  MoveL 1987 to (-124.69, -0.74, -85.2) mm, rotated rx -55.86 ry 0 rz -88.54 deg; joints [-7.765, -84.155, 125.135, -193.916, 25.687, 224.937, -15.943]
  MoveL 1988 to (-128.3, 0.76, -79.65) mm, rotated rx -58.38 ry 0 rz -89.25 deg; joints [-7.042, -84.625, 125.115, -192.318, 25.683, 221.219, -14.624]
  MoveL 1989 to (-129.64, 1.6, -77.44) mm, rotated rx -59.45 ry 0 rz -89.66 deg; joints [-6.738, -84.814, 125.113, -191.644, 25.683, 219.644, -13.978]
  MoveL 1990 to (-130.13, 1.75, -76.61) mm, rotated rx -59.6 ry 0 rz -89.68 deg; joints [-6.67, -84.846, 125.104, -191.491, 25.683, 219.379, -13.911]
  MoveL 1991 to (-131.58, 1.85, -74.08) mm, rotated rx -60.65 ry 0 rz -89.72 deg; joints [-6.348, -85.031, 125.098, -190.776, 25.683, 217.779, -13.631]
  MoveL 1992 to (-131.68, 2.01, -73.92) mm, rotated rx -61.25 ry 0 rz -90 deg; joints [-6.228, -85.122, 125.098, -190.529, 25.626, 216.991, -13.301]
  MoveL 1993 to (-132.47, 3.26, -72.44) mm, rotated rx -61.9 ry 0 rz -90.54 deg; joints [-6.033, -85.23, 125.095, -190.094, 25.626, 216.013, -12.623]
  MoveL 1994 to (-132.84, 3.74, -71.74) mm, rotated rx -62.11 ry 0 rz -90.68 deg; joints [-5.957, -85.258, 125.083, -189.924, 25.626, 215.669, -12.434]
  MoveL 1995 to (-135.12, 6.38, -67.14) mm, rotated rx -64.03 ry 0 rz -91.76 deg; joints [-5.36, -85.56, 125.068, -188.59, 25.626, 212.719, -10.966]
  MoveL 1996 to (-136.66, 9.17, -63.61) mm, rotated rx -65.62 ry 0 rz -92.98 deg; joints [-4.871, -85.803, 125.068, -187.496, 25.624, 210.269, -9.452]
  MoveL 1997 to (-137.15, 9.63, -62.48) mm, rotated rx -65.62 ry 0 rz -92.98 deg; joints [-4.813, -85.796, 125.038, -187.365, 25.624, 210.166, -9.424]
  MoveL 1998 to (-137.46, 9.66, -61.8) mm, rotated rx -65.75 ry 0 rz -92.99 deg; joints [-4.754, -85.823, 125.037, -187.234, 25.624, 209.938, -9.381]
  MoveL 1999 to (-138.91, 9.39, -58.5) mm, rotated rx -67.12 ry 0 rz -92.84 deg; joints [-4.317, -86.01, 125.026, -186.253, 25.624, 207.801, -9.287]
  MoveL 2000 to (-139.18, 9.27, -57.89) mm, rotated rx -67.23 ry 0 rz -92.81 deg; joints [-4.264, -86.035, 125.026, -186.136, 25.62, 207.599, -9.292]
  MoveL 2001 to (-140.3, 7.99, -55.3) mm, rotated rx -68.09 ry 0 rz -92.35 deg; joints [-3.96, -86.17, 125.028, -185.454, 25.619, 206.193, -9.603]
  MoveL 2002 to (-140.85, 7.99, -53.9) mm, rotated rx -69.03 ry 0 rz -92.23 deg; joints [-3.698, -86.248, 125.002, -184.865, 25.619, 204.788, -9.593]
  MoveL 2003 to (-141.12, 7.84, -53.2) mm, rotated rx -69.03 ry 0 rz -92.23 deg; joints [-3.663, -86.268, 125.002, -184.79, 25.601, 204.728, -9.589]
  MoveL 2004 to (-141.46, 7.5, -52.35) mm, rotated rx -69.38 ry 0 rz -92.09 deg; joints [-3.55, -86.309, 124.998, -184.535, 25.601, 204.182, -9.678]
  MoveL 2005 to (-143.81, 3.71, -45.92) mm, rotated rx -71.82 ry 0 rz -90.62 deg; joints [-2.721, -86.589, 124.971, -182.667, 25.601, 200.243, -10.807]
  MoveL 2006 to (-143.79, 3.76, -45.99) mm, rotated rx -72.66 ry 0 rz -90.59 deg; joints [-2.549, -86.63, 124.954, -182.281, 25.601, 199.099, -10.766]
  MoveL 2007 to (-144.66, 5.18, -43.07) mm, rotated rx -73.82 ry 0 rz -91.15 deg; joints [-2.156, -86.735, 124.931, -181.395, 25.601, 197.222, -10.071]
  MoveL 2008 to (-144.92, 5.41, -42.15) mm, rotated rx -73.82 ry 0 rz -91.15 deg; joints [-2.11, -86.73, 124.913, -181.29, 25.601, 197.138, -10.058]
  MoveL 2009 to (-145.17, 5.36, -41.27) mm, rotated rx -73.92 ry 0 rz -91.15 deg; joints [-2.045, -86.751, 124.913, -181.143, 25.601, 196.921, -10.032]
  MoveL 2010 to (-145.6, 4.99, -39.76) mm, rotated rx -75.16 ry 0 rz -91.08 deg; joints [-1.707, -86.843, 124.903, -180.379, 25.601, 195.072, -9.994]
  MoveL 2011 to (-146.32, 6.55, -36.79) mm, rotated rx -76.33 ry 0 rz -91.69 deg; joints [-1.306, -86.925, 124.872, -179.475, 25.601, 193.173, -9.275]
  MoveL 2012 to (-146.5, 7.02, -35.98) mm, rotated rx -76.68 ry 0 rz -91.89 deg; joints [-1.19, -86.95, 124.865, -179.213, 25.601, 192.612, -9.046]
  MoveL 2013 to (-147.72, 11.76, -29.12) mm, rotated rx -79.41 ry 0 rz -93.75 deg; joints [-0.253, -87.095, 124.783, -177.091, 25.601, 188.16, -6.982]
  MoveL 2014 to (-147.89, 15.71, -26.25) mm, rotated rx -80.75 ry 0 rz -95.48 deg; joints [0.184, -87.181, 124.772, -176.101, 25.601, 186.018, -5.174]
  MoveL 2015 to (-147.93, 16.33, -25.65) mm, rotated rx -80.87 ry 0 rz -95.59 deg; joints [0.239, -87.161, 124.744, -175.974, 25.602, 185.797, -5.057]
  MoveL 2016 to (-148.25, 18.54, -22.05) mm, rotated rx -82.08 ry 0 rz -96.3 deg; joints [0.685, -87.163, 124.666, -174.962, 25.602, 183.763, -4.303]
  MoveL 2017 to (-148.41, 18.88, -20.63) mm, rotated rx -82.08 ry 0 rz -96.3 deg; joints [0.757, -87.157, 124.666, -174.808, 25.658, 183.639, -4.256]
  MoveL 2018 to (-148.62, 18.58, -19.38) mm, rotated rx -82.16 ry 0 rz -96.29 deg; joints [0.84, -87.184, 124.675, -174.62, 25.658, 183.398, -4.252]
  MoveL 2019 to (-148.94, 17.65, -17.69) mm, rotated rx -82.81 ry 0 rz -95.93 deg; joints [1.067, -87.189, 124.644, -174.105, 25.658, 182.333, -4.597]
  MoveL 2020 to (-149.44, 16.99, -13.68) mm, rotated rx -84.63 ry 0 rz -95.55 deg; joints [1.669, -87.189, 124.582, -172.757, 25.74, 179.418, -4.882]
  MoveL 2021 to (-149.51, 16.81, -13.05) mm, rotated rx -84.73 ry 0 rz -95.52 deg; joints [1.722, -87.195, 124.58, -172.636, 25.74, 179.223, -4.914]
  MoveL 2022 to (-149.73, 16.26, -10.96) mm, rotated rx -85.58 ry 0 rz -95.28 deg; joints [2.016, -87.196, 124.561, -171.985, 25.796, 177.841, -5.106]
  MoveL 2023 to (-149.72, 16.22, -11.05) mm, rotated rx -86.54 ry 0 rz -95.58 deg; joints [2.223, -87.245, 124.581, -171.514, 25.796, 176.502, -4.798]
  MoveL 2024 to (-149.59, 18.71, -8.96) mm, rotated rx -87.54 ry 0 rz -97 deg; joints [2.553, -87.314, 124.605, -170.766, 25.796, 174.892, -3.374]
  MoveL 2025 to (-148.52, 25.7, -9.48) mm, rotated rx -87.35 ry 0 rz -99.88 deg; joints [2.485, -87.334, 124.605, -170.895, 25.713, 175.184, -0.55]
  MoveL 2026 to (-148.27, 27.19, -9.1) mm, rotated rx -87.35 ry 0 rz -99.88 deg; joints [2.5, -87.245, 124.553, -170.888, 25.806, 175.184, -0.495]
  MoveL 2027 to (-148.17, 27.92, -8.63) mm, rotated rx -87.52 ry 0 rz -100.16 deg; joints [2.563, -87.245, 124.552, -170.752, 25.823, 174.897, -0.204]
  MoveL 2028 to (-147.29, 33.08, -4.1) mm, rotated rx -89.39 ry 0 rz -102.59 deg; joints [3.204, -87.259, 124.508, -169.293, 25.823, 171.845, 2.19]
  MoveL 2029 to (-147.14, 33.77, -4.05) mm, rotated rx -89.41 ry 0 rz -102.85 deg; joints [3.211, -87.259, 124.508, -169.278, 25.826, 171.813, 2.457]
  MoveL 2030 to (-143.96, 45.19, -6.36) mm, rotated rx -88.52 ry 0 rz -107.6 deg; joints [2.899, -87.293, 124.508, -169.925, 25.639, 173.219, 7.097]
  MoveL 2031 to (-142.1, 50.49, -8.11) mm, rotated rx -87.83 ry 0 rz -109.84 deg; joints [2.657, -87.305, 124.508, -170.441, 25.526, 174.326, 9.262]
  MoveL 2032 to (-141.84, 51.2, -8.22) mm, rotated rx -87.83 ry 0 rz -109.84 deg; joints [2.648, -87.25, 124.46, -170.46, 25.526, 174.342, 9.256]
  MoveL 2033 to (-141.67, 51.67, -8.22) mm, rotated rx -87.83 ry 0 rz -110.03 deg; joints [2.649, -87.25, 124.46, -170.459, 25.526, 174.339, 9.45]
  MoveL 2034 to (-139.95, 56.28, -7.34) mm, rotated rx -88.15 ry 0 rz -111.73 deg; joints [2.763, -87.232, 124.46, -170.228, 25.617, 173.839, 11.21]
  MoveL 2035 to (-137.43, 62.13, -7.66) mm, rotated rx -88.04 ry 0 rz -114.37 deg; joints [2.724, -87.256, 124.46, -170.29, 25.534, 173.991, 13.796]
  MoveL 2036 to (-135.16, 66.76, -9.11) mm, rotated rx -87.45 ry 0 rz -116.54 deg; joints [2.522, -87.278, 124.46, -170.71, 25.401, 174.912, 15.878]
  MoveL 2037 to (-134.83, 67.4, -9.2) mm, rotated rx -87.45 ry 0 rz -116.54 deg; joints [2.515, -87.224, 124.413, -170.727, 25.401, 174.926, 15.872]
  MoveL 2038 to (-134.37, 68.32, -9.18) mm, rotated rx -87.46 ry 0 rz -116.93 deg; joints [2.517, -87.224, 124.413, -170.722, 25.402, 174.914, 16.264]
  MoveL 2039 to (-133.91, 69.25, -8.94) mm, rotated rx -87.46 ry 0 rz -116.93 deg; joints [2.527, -87.162, 124.374, -170.718, 25.458, 174.914, 16.297]
  MoveL 2040 to (-130.27, 76.23, -5.17) mm, rotated rx -88.89 ry 0 rz -119.93 deg; joints [3.033, -87.158, 124.374, -169.615, 25.629, 172.594, 19.389]
  MoveL 2041 to (-129.97, 76.76, -4.82) mm, rotated rx -88.98 ry 0 rz -120.08 deg; joints [3.071, -87.149, 124.374, -169.542, 25.667, 172.446, 19.565]
  MoveL 2042 to (-128.21, 79.76, -2.85) mm, rotated rx -89.74 ry 0 rz -121.42 deg; joints [3.338, -87.142, 124.374, -168.964, 25.756, 171.222, 20.946]
  MoveL 2043 to (-127.99, 80.12, -2.6) mm, rotated rx -89.83 ry 0 rz -121.57 deg; joints [3.37, -87.14, 124.374, -168.895, 25.77, 171.077, 21.109]
  MoveL 2044 to (-126.08, 83.14, -0.8) mm, rotated rx -90.54 ry 0 rz -122.97 deg; joints [3.618, -87.132, 124.374, -168.36, 25.847, 169.935, 22.541]
  MoveL 2045 to (-125.78, 83.59, -0.43) mm, rotated rx -90.54 ry 0 rz -122.97 deg; joints [3.636, -87.11, 124.374, -168.347, 25.919, 169.93, 22.588]
  MoveL 2046 to (-125.56, 83.91, -0.09) mm, rotated rx -90.67 ry 0 rz -123.12 deg; joints [3.682, -87.107, 124.374, -168.249, 25.936, 169.721, 22.74]
  MoveL 2047 to (-125.22, 84.42, 0.77) mm, rotated rx -90.67 ry 0 rz -123.12 deg; joints [3.725, -87.079, 124.374, -168.189, 26.026, 169.679, 22.797]
  MoveL 2048 to (-124.21, 85.78, 4.61) mm, rotated rx -92.13 ry 0 rz -123.76 deg; joints [4.24, -87.039, 124.374, -167.109, 26.227, 167.36, 23.512]
  MoveL 2049 to (-121.27, 89.62, 8.28) mm, rotated rx -93.9 ry 0 rz -125.89 deg; joints [4.815, -87.007, 124.374, -165.88, 26.374, 164.611, 25.651]
  MoveL 2050 to (-120.98, 89.99, 8.63) mm, rotated rx -94.04 ry 0 rz -126.08 deg; joints [4.863, -87.002, 124.374, -165.779, 26.391, 164.389, 25.845]
  MoveL 2051 to (-117.7, 93.74, 12.84) mm, rotated rx -95.6 ry 0 rz -127.92 deg; joints [5.418, -86.916, 124.374, -164.664, 26.653, 161.95, 27.751]
  MoveL 2052 to (-117.06, 94.32, 14.38) mm, rotated rx -95.6 ry 0 rz -127.92 deg; joints [5.493, -86.869, 124.374, -164.564, 26.789, 161.881, 27.828]
  MoveL 2053 to (-116.97, 94.28, 15.39) mm, rotated rx -95.69 ry 0 rz -127.93 deg; joints [5.564, -86.857, 124.374, -164.423, 26.819, 161.68, 27.845]
  MoveL 2054 to (-117, 93.95, 17.04) mm, rotated rx -96.32 ry 0 rz -127.82 deg; joints [5.785, -86.818, 124.374, -163.985, 26.921, 160.707, 27.755]
  MoveL 2055 to (-116.24, 94.53, 18.96) mm, rotated rx -97.62 ry 0 rz -128.26 deg; joints [6.165, -86.752, 124.374, -163.228, 27.078, 158.815, 28.197]
  MoveL 2056 to (-115.96, 94.57, 20.45) mm, rotated rx -97.62 ry 0 rz -128.26 deg; joints [6.239, -86.728, 124.374, -163.097, 27.139, 158.716, 28.219]
  MoveL 2057 to (-116.14, 94.01, 21.92) mm, rotated rx -97.76 ry 0 rz -128.23 deg; joints [6.344, -86.728, 124.378, -162.865, 27.139, 158.394, 28.166]
  MoveL 2058 to (-117.02, 92.32, 24.27) mm, rotated rx -99.1 ry 0 rz -127.32 deg; joints [6.75, -86.614, 124.378, -162.121, 27.401, 156.492, 27.315]
  MoveL 2059 to (-116.98, 92.03, 25.56) mm, rotated rx -99.59 ry 0 rz -127.24 deg; joints [6.921, -86.572, 124.378, -161.796, 27.489, 155.748, 27.239]
  MoveL 2060 to (-117.05, 91.68, 26.5) mm, rotated rx -99.75 ry 0 rz -127.18 deg; joints [7.002, -86.558, 124.378, -161.633, 27.513, 155.466, 27.165]
  MoveL 2061 to (-117.17, 90.63, 29.37) mm, rotated rx -100.93 ry 0 rz -126.8 deg; joints [7.4, -86.447, 124.378, -160.896, 27.731, 153.722, 26.798]
  MoveL 2062 to (-116.45, 90.99, 31.12) mm, rotated rx -102.26 ry 0 rz -127.11 deg; joints [7.769, -86.342, 124.378, -160.212, 27.922, 151.885, 27.102]
  MoveL 2063 to (-116.16, 91, 32.15) mm, rotated rx -102.26 ry 0 rz -127.11 deg; joints [7.82, -86.319, 124.38, -160.136, 27.975, 151.832, 27.119]
  MoveL 2064 to (-116.09, 90.62, 33.43) mm, rotated rx -103.42 ry 0 rz -127.24 deg; joints [8.131, -86.245, 124.38, -159.527, 28.074, 150.208, 27.201]
  MoveL 2065 to (-114.95, 91.49, 34.97) mm, rotated rx -104.01 ry 0 rz -127.78 deg; joints [8.333, -86.178, 124.38, -159.165, 28.189, 149.343, 27.736]
  MoveL 2066 to (-114.26, 91.74, 36.56) mm, rotated rx -104.01 ry 0 rz -127.78 deg; joints [8.41, -86.125, 124.38, -159.076, 28.307, 149.289, 27.785]
  MoveL 2067 to (-114.19, 91.07, 38.4) mm, rotated rx -104.17 ry 0 rz -127.78 deg; joints [8.537, -86.101, 124.38, -158.814, 28.322, 148.929, 27.74]
  MoveL 2068 to (-115.08, 88.3, 42.05) mm, rotated rx -105.61 ry 0 rz -126.7 deg; joints [9.018, -85.922, 124.38, -157.975, 28.604, 146.879, 26.63]
  MoveL 2069 to (-115.21, 87.18, 43.98) mm, rotated rx -106.52 ry 0 rz -126.22 deg; joints [9.3, -85.801, 124.38, -157.51, 28.8, 145.643, 26.156]
  MoveL 2070 to (-115.3, 86.78, 44.52) mm, rotated rx -106.52 ry 0 rz -126.22 deg; joints [9.33, -85.813, 124.395, -157.446, 28.8, 145.594, 26.143]
  MoveL 2071 to (-115.4, 86.48, 44.85) mm, rotated rx -106.64 ry 0 rz -126.1 deg; joints [9.373, -85.795, 124.395, -157.374, 28.825, 145.413, 26.019]
  MoveL 2072 to (-116.47, 83.68, 47.31) mm, rotated rx -107.55 ry 0 rz -125.03 deg; joints [9.681, -85.674, 124.395, -156.836, 28.989, 144.121, 24.905]
  MoveL 2073 to (-116.37, 82.67, 49.3) mm, rotated rx -108.7 ry 0 rz -124.46 deg; joints [10.011, -85.5, 124.395, -156.344, 29.271, 142.643, 24.356]
  MoveL 2074 to (-116.42, 82.21, 49.94) mm, rotated rx -108.7 ry 0 rz -124.46 deg; joints [10.046, -85.509, 124.41, -156.272, 29.271, 142.588, 24.339]
  MoveL 2075 to (-116.6, 81.61, 50.52) mm, rotated rx -108.79 ry 0 rz -124.38 deg; joints [10.095, -85.509, 124.42, -156.168, 29.272, 142.418, 24.231]
  MoveL 2076 to (-117.58, 78.88, 52.54) mm, rotated rx -109.6 ry 0 rz -123.24 deg; joints [10.358, -85.385, 124.42, -155.739, 29.438, 141.308, 23.062]
  MoveL 2077 to (-117.87, 77.18, 54.39) mm, rotated rx -110.51 ry 0 rz -122.43 deg; joints [10.629, -85.234, 124.42, -155.341, 29.661, 140.142, 22.249]
  MoveL 2078 to (-118.08, 76.44, 54.96) mm, rotated rx -110.51 ry 0 rz -122.43 deg; joints [10.664, -85.268, 124.457, -155.268, 29.661, 140.087, 22.234]
  MoveL 2079 to (-118.37, 75.77, 55.27) mm, rotated rx -110.56 ry 0 rz -122.33 deg; joints [10.694, -85.283, 124.477, -155.205, 29.661, 139.985, 22.112]
  MoveL 2080 to (-119.55, 73.3, 56.05) mm, rotated rx -110.88 ry 0 rz -121.21 deg; joints [10.795, -85.231, 124.477, -155.044, 29.728, 139.557, 20.984]
  MoveL 2081 to (-119.75, 72.81, 56.26) mm, rotated rx -110.99 ry 0 rz -120.91 deg; joints [10.828, -85.206, 124.477, -155.012, 29.774, 139.428, 20.698]
  MoveL 2082 to (-120.75, 68.2, 59.75) mm, rotated rx -112.58 ry 0 rz -118.8 deg; joints [11.308, -84.921, 124.477, -154.318, 30.165, 137.402, 18.558]
  MoveL 2083 to (-120.68, 68.16, 59.97) mm, rotated rx -113.09 ry 0 rz -118.48 deg; joints [11.417, -84.827, 124.477, -154.221, 30.331, 136.843, 18.287]
  MoveL 2084 to (-119.88, 66.14, 63.73) mm, rotated rx -114.66 ry 0 rz -117.9 deg; joints [11.903, -84.546, 124.478, -153.484, 30.655, 134.802, 17.604]
  MoveL 2085 to (-119.8, 65.76, 64.28) mm, rotated rx -114.66 ry 0 rz -117.9 deg; joints [11.931, -84.547, 124.487, -153.426, 30.655, 134.76, 17.585]
  MoveL 2086 to (-119.77, 65.42, 64.66) mm, rotated rx -114.82 ry 0 rz -117.78 deg; joints [11.982, -84.516, 124.487, -153.352, 30.689, 134.549, 17.453]
  MoveL 2087 to (-119.95, 61.76, 67.86) mm, rotated rx -116.05 ry 0 rz -116.47 deg; joints [12.369, -84.288, 124.487, -152.752, 30.919, 132.945, 16.034]
  MoveL 2088 to (-120.08, 60.96, 68.35) mm, rotated rx -116.05 ry 0 rz -116.47 deg; joints [12.401, -84.322, 124.526, -152.688, 30.919, 132.897, 16.018]
  MoveL 2089 to (-120.24, 60.38, 68.59) mm, rotated rx -116.15 ry 0 rz -116.22 deg; joints [12.432, -84.303, 124.528, -152.644, 30.944, 132.768, 15.76]
  MoveL 2090 to (-120.98, 56.47, 70.56) mm, rotated rx -117.04 ry 0 rz -114.49 deg; joints [12.694, -84.125, 124.533, -152.289, 31.154, 131.674, 13.981]
  MoveL 2091 to (-118.84, 57.87, 73.02) mm, rotated rx -119.86 ry 0 rz -115.85 deg; joints [13.333, -83.729, 124.533, -151.276, 31.47, 128.216, 15.064]
  MoveL 2092 to (-117.93, 59.53, 73.19) mm, rotated rx -119.93 ry 0 rz -116.68 deg; joints [13.355, -83.714, 124.533, -151.246, 31.484, 128.126, 15.881]
  MoveL 2093 to (-116.76, 60.86, 73.96) mm, rotated rx -119.96 ry 0 rz -116.69 deg; joints [13.377, -83.573, 124.441, -151.246, 31.536, 128.115, 15.894]
  MoveL 2094 to (-115.68, 60.98, 75.54) mm, rotated rx -119.99 ry 0 rz -116.7 deg; joints [13.455, -83.49, 124.441, -151.193, 31.66, 128.079, 15.93]
  MoveL 2095 to (-115.1, 60.65, 76.68) mm, rotated rx -120.49 ry 0 rz -116.68 deg; joints [13.606, -83.402, 124.486, -151.051, 31.848, 127.523, 15.93]
  MoveL 2096 to (-114.03, 60.99, 78.01) mm, rotated rx -121.53 ry 0 rz -117.15 deg; joints [13.854, -83.226, 124.487, -150.681, 31.986, 126.268, 16.281]
  MoveL 2097 to (-113.32, 60.92, 79.08) mm, rotated rx -121.53 ry 0 rz -117.15 deg; joints [13.904, -83.176, 124.487, -150.639, 32.053, 126.256, 16.285]
  MoveL 2098 to (-112.82, 60.37, 80.21) mm, rotated rx -121.68 ry 0 rz -117.14 deg; joints [13.991, -83.14, 124.527, -150.557, 32.161, 126.074, 16.285]
  MoveL 2099 to (-111.85, 57.98, 83.26) mm, rotated rx -123.17 ry 0 rz -116.42 deg; joints [14.421, -82.89, 124.706, -150.237, 32.786, 124.52, 15.672]
  MoveL 2100 to (-109.17, 56.99, 87.4) mm, rotated rx -125.32 ry 0 rz -116.53 deg; joints [14.983, -82.416, 124.727, -149.536, 33.225, 122.038, 15.56]
  MoveL 2101 to (-108.53, 56, 88.83) mm, rotated rx -125.32 ry 0 rz -116.53 deg; joints [15.062, -82.405, 124.784, -149.46, 33.314, 122.01, 15.56]
  MoveL 2102 to (-108.42, 55.2, 89.47) mm, rotated rx -125.62 ry 0 rz -116.21 deg; joints [15.148, -82.344, 124.818, -149.403, 33.443, 121.699, 15.253]
  MoveL 2103 to (-108.75, 53.37, 90.18) mm, rotated rx -125.62 ry 0 rz -116.21 deg; joints [15.205, -82.43, 124.916, -149.296, 33.443, 121.625, 15.22]
  MoveL 2104 to (-112.59, 43.93, 90.56) mm, rotated rx -125.9 ry 0 rz -111.26 deg; joints [15.267, -82.365, 124.924, -149.254, 33.534, 121.353, 10.279]
  MoveL 2105 to (-113.25, 41.96, 90.66) mm, rotated rx -125.95 ry 0 rz -110.24 deg; joints [15.281, -82.349, 124.925, -149.245, 33.554, 121.3, 9.264]
  MoveL 2106 to (-113.56, 41.16, 90.65) mm, rotated rx -125.94 ry 0 rz -109.98 deg; joints [15.283, -82.372, 124.944, -149.241, 33.554, 121.306, 9.002]
  MoveL 2107 to (-113.92, 38.56, 91.31) mm, rotated rx -126.3 ry 0 rz -108.36 deg; joints [15.369, -82.25, 124.944, -149.215, 33.721, 120.978, 7.418]
  MoveL 2108 to (-113.89, 38.54, 91.36) mm, rotated rx -127.16 ry 0 rz -107.51 deg; joints [15.503, -82.032, 124.935, -149.215, 34.026, 120.2, 6.642]
  MoveL 2109 to (-112.68, 37.99, 93.08) mm, rotated rx -128.64 ry 0 rz -107.68 deg; joints [15.823, -81.751, 124.935, -148.756, 34.175, 118.492, 6.59]
  MoveL 2110 to (-110.37, 39.47, 95.21) mm, rotated rx -129.67 ry 0 rz -108.71 deg; joints [16.083, -81.492, 124.935, -148.43, 34.35, 117.33, 7.458]
  MoveL 2111 to (-108.12, 42.41, 96.54) mm, rotated rx -130.58 ry 0 rz -110.86 deg; joints [16.289, -81.324, 124.935, -148.082, 34.373, 116.225, 9.388]
  MoveL 2112 to (-122.31, 47.82, 109.55) mm, rotated rx -130.58 ry 0 rz -110.86 deg; joints [17.015, -81.832, 124.935, -147.724, 35.769, 115.928, 11.072]
  Set speed (1000.0 mm/s)
  MoveL 2113 to (-119.4, 45.41, 113.71) mm, rotated rx -130.84 ry 0 rz -110.73 deg; joints [17.251, -81.623, 124.936, -147.355, 35.823, 115.48, 10.707]
  Set speed (5.0 mm/s)
  MoveL 2114 to (-105.24, 40.05, 100.63) mm, rotated rx -130.84 ry 0 rz -110.73 deg; joints [16.522, -81.126, 124.933, -147.685, 34.394, 115.748, 9.003]
  Set speed (16.7 mm/s)
  MoveL 2115 to (-106.36, 36.25, 100.88) mm, rotated rx -130.97 ry 0 rz -108.71 deg; joints [16.557, -81.101, 124.96, -147.684, 34.47, 115.642, 7.009]
  MoveL 2116 to (-120.67, 41.09, 113.99) mm, rotated rx -130.97 ry 0 rz -108.71 deg; joints [17.287, -81.594, 124.96, -147.351, 35.898, 115.372, 8.711]
  Set speed (1000.0 mm/s)
  MoveL 2117 to (-118.91, 26.12, 120.09) mm, rotated rx -134.04 ry 0 rz -101.52 deg; joints [18.009, -80.673, 124.96, -146.703, 36.636, 112.216, 1.177]
  Set speed (5.0 mm/s)
  MoveL 2118 to (-104.82, 23.25, 106.19) mm, rotated rx -134.04 ry 0 rz -101.52 deg; joints [17.246, -80.243, 124.96, -147.004, 35.105, 112.431, -0.563]
  Set speed (16.7 mm/s)
  MoveL 2119 to (-104.41, 21.99, 106.87) mm, rotated rx -134.42 ry 0 rz -100.89 deg; joints [17.341, -80.162, 125.024, -146.997, 35.3, 112.12, -1.156]
  MoveL 2120 to (-102.69, 19.1, 109.07) mm, rotated rx -135.76 ry 0 rz -99.29 deg; joints [17.628, -79.797, 125.032, -146.697, 35.53, 110.72, -2.963]
  MoveL 2121 to (-102.33, 17.43, 109.68) mm, rotated rx -135.76 ry 0 rz -99.29 deg; joints [17.679, -79.866, 125.12, -146.607, 35.53, 110.665, -3.002]
  MoveL 2122 to (-102.37, 16.88, 109.73) mm, rotated rx -135.79 ry 0 rz -98.98 deg; joints [17.685, -79.858, 125.123, -146.605, 35.542, 110.64, -3.312]
  MoveL 2123 to (-102.11, 14.05, 110.35) mm, rotated rx -136.17 ry 0 rz -97.19 deg; joints [17.764, -79.733, 125.125, -146.565, 35.655, 110.28, -5.136]
  MoveL 2124 to (-102.17, 14.13, 110.3) mm, rotated rx -137.24 ry 0 rz -96.25 deg; joints [17.893, -79.461, 125.103, -146.565, 35.92, 109.327, -6.068]
  MoveL 2125 to (-99.55, 14.42, 112.66) mm, rotated rx -138.55 ry 0 rz -96.54 deg; joints [18.172, -79.095, 125.104, -146.222, 36.066, 107.922, -6.066]
  MoveL 2126 to (-97.81, 15.28, 114.06) mm, rotated rx -139.93 ry 0 rz -97.63 deg; joints [18.416, -78.817, 125.109, -145.827, 36.066, 106.38, -5.341]
  MoveL 2127 to (-95.33, 17.87, 115.77) mm, rotated rx -140.85 ry 0 rz -99.27 deg; joints [18.607, -78.545, 125.109, -145.593, 36.155, 105.406, -3.922]
  MoveL 2128 to (-94.23, 18.44, 116.58) mm, rotated rx -140.85 ry 0 rz -99.27 deg; joints [18.631, -78.445, 125.063, -145.563, 36.162, 105.406, -3.973]
  MoveL 2129 to (-93.66, 18.46, 117.03) mm, rotated rx -140.94 ry 0 rz -99.3 deg; joints [18.662, -78.399, 125.065, -145.533, 36.184, 105.318, -3.973]
  MoveL 2130 to (-92.1, 18.26, 118.3) mm, rotated rx -141.72 ry 0 rz -99.34 deg; joints [18.83, -78.203, 125.157, -145.482, 36.458, 104.634, -3.973]
  MoveL 2131 to (-89.1, 18.17, 120.59) mm, rotated rx -143.24 ry 0 rz -99.6 deg; joints [19.12, -77.798, 125.206, -145.184, 36.651, 103.104, -4.028]
  MoveL 2132 to (-88, 17.68, 121.46) mm, rotated rx -143.24 ry 0 rz -99.6 deg; joints [19.165, -77.76, 125.234, -145.139, 36.684, 103.102, -4.07]
  MoveL 2133 to (-87.65, 17.34, 121.76) mm, rotated rx -143.43 ry 0 rz -99.42 deg; joints [19.203, -77.707, 125.242, -145.105, 36.713, 102.909, -4.29]
  MoveL 2134 to (-87.09, 16.45, 122.28) mm, rotated rx -143.43 ry 0 rz -99.42 deg; joints [19.238, -77.723, 125.287, -145.047, 36.713, 102.882, -4.331]
  MoveL 2135 to (-85.63, 12.54, 123.76) mm, rotated rx -144.42 ry 0 rz -96.96 deg; joints [19.423, -77.447, 125.326, -144.879, 36.855, 101.914, -6.998]
  MoveL 2136 to (-84.87, 11.35, 124.41) mm, rotated rx -144.96 ry 0 rz -95.98 deg; joints [19.509, -77.287, 125.327, -144.803, 36.922, 101.392, -8.081]
  MoveL 2137 to (-84.51, 10.45, 124.72) mm, rotated rx -144.96 ry 0 rz -95.98 deg; joints [19.537, -77.32, 125.377, -144.757, 36.922, 101.369, -8.107]
  MoveL 2138 to (-84.4, 9.74, 124.85) mm, rotated rx -145.01 ry 0 rz -95.79 deg; joints [19.554, -77.33, 125.401, -144.73, 36.922, 101.313, -8.323]
  MoveL 2139 to (-84.29, 8.18, 125.03) mm, rotated rx -145.13 ry 0 rz -94.72 deg; joints [19.577, -77.295, 125.411, -144.721, 36.953, 101.208, -9.404]
  MoveL 2140 to (-84.32, 8.21, 125.03) mm, rotated rx -145.76 ry 0 rz -93.43 deg; joints [19.619, -77.062, 125.321, -144.721, 37.02, 100.633, -10.763]
  MoveL 2141 to (-83.75, 7.93, 125.43) mm, rotated rx -146.04 ry 0 rz -93.26 deg; joints [19.667, -76.985, 125.325, -144.661, 37.034, 100.351, -11.009]
  MoveL 2142 to (-83.33, 7.67, 125.72) mm, rotated rx -146.1 ry 0 rz -93.21 deg; joints [19.689, -76.963, 125.335, -144.629, 37.036, 100.28, -11.104]
  MoveL 2143 to (-82.15, 6.44, 126.56) mm, rotated rx -146.53 ry 0 rz -92.57 deg; joints [19.781, -76.846, 125.374, -144.54, 37.095, 99.856, -11.855]
  MoveL 2144 to (-81.38, 6.16, 127.08) mm, rotated rx -147.23 ry 0 rz -92.07 deg; joints [19.873, -76.66, 125.374, -144.461, 37.162, 99.191, -12.482]
  MoveL 2145 to (-80.87, 5.85, 127.42) mm, rotated rx -147.23 ry 0 rz -92.07 deg; joints [19.894, -76.655, 125.396, -144.439, 37.174, 99.188, -12.502]
  MoveL 2146 to (-80.53, 5.57, 127.65) mm, rotated rx -147.39 ry 0 rz -91.87 deg; joints [19.921, -76.609, 125.399, -144.404, 37.179, 99.02, -12.747]
  MoveL 2147 to (-78.37, 3.33, 129.04) mm, rotated rx -148.32 ry 0 rz -90.39 deg; joints [20.09, -76.357, 125.469, -144.269, 37.316, 98.147, -14.435]
  MoveL 2148 to (-88.88, 3.4, 146.06) mm, rotated rx -148.32 ry 0 rz -90.39 deg; joints [20.959, -76.423, 125.373, -144.051, 39.145, 98.147, -12.66]
  Set speed (1000.0 mm/s)
  MoveL 2149 to (-85.2, 1.1, 148.27) mm, rotated rx -149.48 ry 0 rz -90 deg; joints [21.198, -76.142, 125.476, -143.716, 39.146, 96.927, -13.492]
  Set speed (5.0 mm/s)
  MoveL 2150 to (-75.05, 1.1, 131.04) mm, rotated rx -149.48 ry 0 rz -90 deg; joints [20.326, -76.113, 125.598, -143.946, 37.337, 96.927, -15.233]
  Set speed (16.7 mm/s)
  MoveL 2151 to (-74.99, 0.23, 131.08) mm, rotated rx -149.51 ry 0 rz -89.33 deg; joints [20.33, -76.104, 125.601, -143.946, 37.345, 96.905, -15.908]
  MoveL 2152 to (-75.02, -0.11, 131.07) mm, rotated rx -149.73 ry 0 rz -87.95 deg; joints [20.327, -75.972, 125.518, -143.961, 37.345, 96.712, -17.327]
  MoveL 2153 to (-73.47, -2, 131.92) mm, rotated rx -149.99 ry 0 rz -87.96 deg; joints [20.425, -75.985, 125.642, -143.814, 37.345, 96.396, -17.458]
  MoveL 2154 to (-72.96, -2.95, 132.2) mm, rotated rx -149.99 ry 0 rz -87.96 deg; joints [20.453, -76.026, 125.701, -143.768, 37.345, 96.375, -17.485]
  MoveL 2155 to (-72.33, -5.36, 132.45) mm, rotated rx -150.41 ry 0 rz -85.29 deg; joints [20.493, -75.876, 125.677, -143.768, 37.407, 96.02, -20.214]
  MoveL 2156 to (-71.43, -6.39, 132.9) mm, rotated rx -150.78 ry 0 rz -84.4 deg; joints [20.556, -75.779, 125.726, -143.768, 37.518, 95.721, -21.14]
  MoveL 2157 to (-70.8, -7.68, 133.18) mm, rotated rx -150.78 ry 0 rz -84.4 deg; joints [20.592, -75.844, 125.807, -143.71, 37.518, 95.692, -21.169]
  MoveL 2158 to (-70.31, -9.65, 133.31) mm, rotated rx -150.89 ry 0 rz -82.76 deg; joints [20.611, -75.813, 125.822, -143.71, 37.551, 95.596, -22.816]
  MoveL 2159 to (-70.2, -10.42, 133.32) mm, rotated rx -150.9 ry 0 rz -82.61 deg; joints [20.622, -75.849, 125.856, -143.691, 37.551, 95.576, -22.975]
  MoveL 2160 to (-70.14, -12.43, 133.18) mm, rotated rx -150.79 ry 0 rz -80.96 deg; joints [20.605, -75.876, 125.851, -143.714, 37.551, 95.684, -24.584]
  MoveL 2161 to (-69.55, -15.84, 133.12) mm, rotated rx -150.75 ry 0 rz -77.95 deg; joints [20.593, -75.869, 125.832, -143.731, 37.551, 95.729, -27.582]
  MoveL 2162 to (-69.76, -17.49, 132.81) mm, rotated rx -150.75 ry 0 rz -77.95 deg; joints [20.606, -75.996, 125.923, -143.702, 37.551, 95.697, -27.555]
  MoveL 2163 to (-70.51, -19.37, 132.15) mm, rotated rx -150.01 ry 0 rz -75.72 deg; joints [20.484, -76.103, 125.837, -143.874, 37.551, 96.477, -29.563]
  MoveL 2164 to (-70.5, -20.09, 132.05) mm, rotated rx -149.98 ry 0 rz -75.52 deg; joints [20.485, -76.144, 125.862, -143.87, 37.551, 96.491, -29.754]
  MoveL 2165 to (-70.76, -22.23, 131.56) mm, rotated rx -149.53 ry 0 rz -73.12 deg; joints [20.399, -76.191, 125.788, -143.994, 37.55, 96.98, -32.01]
  MoveL 2166 to (-70.5, -23, 131.56) mm, rotated rx -149.53 ry 0 rz -72.49 deg; joints [20.4, -76.189, 125.788, -143.994, 37.552, 96.974, -32.637]
  MoveL 2167 to (-70.37, -23.62, 131.53) mm, rotated rx -149.53 ry 0 rz -72.49 deg; joints [20.409, -76.233, 125.825, -143.977, 37.552, 96.961, -32.635]
  MoveL 2168 to (-70.33, -24.58, 131.38) mm, rotated rx -149.5 ry 0 rz -72.2 deg; joints [20.408, -76.287, 125.856, -143.974, 37.552, 96.987, -32.912]
  MoveL 2169 to (-70.61, -28.42, 130.45) mm, rotated rx -148.78 ry 0 rz -69.44 deg; joints [20.294, -76.477, 125.838, -144.131, 37.552, 97.715, -35.436]
  MoveL 2170 to (-70.7, -29.36, 130.19) mm, rotated rx -148.72 ry 0 rz -69.17 deg; joints [20.283, -76.54, 125.859, -144.131, 37.536, 97.763, -35.678]
  MoveL 2171 to (-71.43, -32.36, 129.07) mm, rotated rx -147.88 ry 0 rz -67.27 deg; joints [20.147, -76.77, 125.846, -144.322, 37.536, 98.632, -37.314]
  MoveL 2172 to (-81.24, -36.47, 146.01) mm, rotated rx -147.88 ry 0 rz -67.27 deg; joints [21.017, -76.838, 125.758, -144.106, 39.374, 98.632, -35.535]
  Set speed (1000.0 mm/s)
  MoveL 2173 to (-77.22, -38.49, 147.66) mm, rotated rx -148.8 ry 0 rz -64.18 deg; joints [21.173, -76.467, 125.758, -144.045, 39.577, 97.844, -38.795]
  Set speed (5.0 mm/s)
  MoveL 2174 to (-67.89, -33.98, 130.56) mm, rotated rx -148.8 ry 0 rz -64.18 deg; joints [20.299, -76.424, 125.861, -144.27, 37.741, 97.844, -40.562]
  Set speed (16.7 mm/s)
  MoveL 2175 to (-67.23, -36.01, 130.36) mm, rotated rx -148.65 ry 0 rz -62.56 deg; joints [20.275, -76.464, 125.857, -144.304, 37.741, 97.998, -42.129]
  MoveL 2176 to (-67.2, -37.94, 129.81) mm, rotated rx -148.3 ry 0 rz -60.2 deg; joints [20.191, -76.472, 125.766, -144.429, 37.741, 98.383, -44.371]
  MoveL 2177 to (-66.35, -38.67, 130.04) mm, rotated rx -148.47 ry 0 rz -59.4 deg; joints [20.218, -76.423, 125.767, -144.392, 37.741, 98.205, -45.227]
  MoveL 2178 to (-65.37, -39.02, 130.42) mm, rotated rx -148.93 ry 0 rz -58.29 deg; joints [20.276, -76.273, 125.767, -144.385, 37.834, 97.815, -46.386]
  MoveL 2179 to (-64.59, -39.53, 130.67) mm, rotated rx -148.93 ry 0 rz -58.29 deg; joints [20.302, -76.31, 125.818, -144.345, 37.834, 97.796, -46.41]
  MoveL 2180 to (-64.18, -39.97, 130.74) mm, rotated rx -148.94 ry 0 rz -58.22 deg; joints [20.314, -76.334, 125.848, -144.324, 37.834, 97.773, -46.492]
  MoveL 2181 to (-63.7, -40.59, 130.77) mm, rotated rx -148.97 ry 0 rz -57.62 deg; joints [20.319, -76.325, 125.848, -144.318, 37.835, 97.74, -47.098]
  MoveL 2182 to (-62.85, -41.02, 131.05) mm, rotated rx -149.31 ry 0 rz -56.23 deg; joints [20.352, -76.181, 125.812, -144.318, 37.886, 97.448, -48.545]
  MoveL 2183 to (-61.73, -42.25, 131.2) mm, rotated rx -149.31 ry 0 rz -56.23 deg; joints [20.386, -76.275, 125.91, -144.26, 37.886, 97.413, -48.562]
  MoveL 2184 to (-61.42, -43.97, 130.78) mm, rotated rx -149.03 ry 0 rz -54.03 deg; joints [20.317, -76.275, 125.829, -144.363, 37.886, 97.728, -50.658]
  MoveL 2185 to (-60.94, -44.4, 130.86) mm, rotated rx -149.05 ry 0 rz -53.95 deg; joints [20.331, -76.299, 125.86, -144.34, 37.886, 97.702, -50.755]
  MoveL 2186 to (-60.17, -45.41, 130.87) mm, rotated rx -149.05 ry 0 rz -53.22 deg; joints [20.337, -76.318, 125.879, -144.33, 37.886, 97.692, -51.484]
  MoveL 2187 to (-58.97, -46.12, 131.16) mm, rotated rx -149.35 ry 0 rz -51.47 deg; joints [20.366, -76.179, 125.84, -144.33, 37.93, 97.436, -53.289]
  MoveL 2188 to (-57.34, -45.99, 131.92) mm, rotated rx -149.74 ry 0 rz -50.8 deg; joints [20.44, -76.053, 125.852, -144.23, 37.93, 97.039, -54.113]
  MoveL 2189 to (-55.9, -47.06, 132.17) mm, rotated rx -150.12 ry 0 rz -50.11 deg; joints [20.503, -76.022, 125.91, -144.14, 37.931, 96.633, -54.904]
  MoveL 2190 to (-53.58, -50.2, 131.97) mm, rotated rx -149.97 ry 0 rz -47.08 deg; joints [20.479, -76.066, 125.907, -144.171, 37.931, 96.789, -57.888]
  MoveL 2191 to (-52.99, -49.57, 132.45) mm, rotated rx -151.13 ry 0 rz -44.97 deg; joints [20.576, -75.653, 125.821, -144.171, 38.081, 95.768, -60.157]
  MoveL 2192 to (-52.53, -49.31, 132.73) mm, rotated rx -151.19 ry 0 rz -44.95 deg; joints [20.597, -75.627, 125.831, -144.143, 38.081, 95.704, -60.218]
  MoveL 2193 to (-49.78, -48.12, 134.21) mm, rotated rx -152.41 ry 0 rz -44.03 deg; joints [20.777, -75.295, 125.869, -143.91, 38.081, 94.49, -61.535]
  MoveL 2194 to (-48.98, -47.93, 134.58) mm, rotated rx -152.41 ry 0 rz -44.03 deg; joints [20.801, -75.293, 125.9, -143.875, 38.082, 94.482, -61.573]
  MoveL 2195 to (-47.83, -48.01, 134.96) mm, rotated rx -152.53 ry 0 rz -43.81 deg; joints [20.84, -75.28, 125.943, -143.821, 38.082, 94.353, -61.858]
  MoveL 2196 to (-46.35, -49.06, 135.1) mm, rotated rx -152.53 ry 0 rz -43.81 deg; joints [20.878, -75.384, 126.051, -143.758, 38.082, 94.316, -61.876]
  MoveL 2197 to (-44.24, -51.83, 134.77) mm, rotated rx -152.25 ry 0 rz -40.91 deg; joints [20.837, -75.458, 126.04, -143.811, 38.082, 94.591, -64.692]
  MoveL 2198 to (-50.34, -58.87, 152.47) mm, rotated rx -152.25 ry 0 rz -40.91 deg; joints [21.72, -75.408, 125.877, -143.549, 39.884, 94.591, -62.995]
  Set speed (1000.0 mm/s)
  MoveL 2199 to (-44.65, -61.37, 153.25) mm, rotated rx -153.05 ry 0 rz -34.75 deg; joints [21.794, -75.057, 125.802, -143.549, 39.992, 93.917, -69.304]
  Set speed (5.0 mm/s)
  MoveL 2200 to (-39.49, -53.92, 135.43) mm, rotated rx -153.05 ry 0 rz -34.75 deg; joints [20.909, -75.125, 125.974, -143.818, 38.192, 93.917, -70.992]
  Set speed (16.7 mm/s)
  MoveL 2201 to (-37.74, -54.13, 135.84) mm, rotated rx -153.16 ry 0 rz -34.49 deg; joints [20.959, -75.153, 126.057, -143.744, 38.192, 93.786, -71.316]
  MoveL 2202 to (-36.32, -54.77, 135.96) mm, rotated rx -153.27 ry 0 rz -33.16 deg; joints [20.975, -75.123, 126.062, -143.726, 38.193, 93.679, -72.685]
  MoveL 2203 to (-41.25, -62.3, 153.82) mm, rotated rx -153.27 ry 0 rz -33.16 deg; joints [21.86, -75.046, 125.883, -143.453, 39.986, 93.679, -71.007]
  Set speed (1000.0 mm/s)
  MoveL 2204 to (-38.06, -61.38, 155.02) mm, rotated rx -154.24 ry 0 rz -31.11 deg; joints [21.99, -74.737, 125.889, -143.298, 39.987, 92.744, -73.382]
  Set speed (5.0 mm/s)
  MoveL 2205 to (-33.57, -53.93, 137.01) mm, rotated rx -154.24 ry 0 rz -31.11 deg; joints [21.103, -74.839, 126.084, -143.581, 38.207, 92.744, -75.038]
  Set speed (16.7 mm/s)
  MoveL 2206 to (-29.71, -54.62, 137.63) mm, rotated rx -154.81 ry 0 rz -27.73 deg; joints [21.181, -74.687, 126.112, -143.488, 38.208, 92.195, -78.613]
  MoveL 2207 to (-27.31, -54.41, 138.2) mm, rotated rx -155.44 ry 0 rz -25.68 deg; joints [21.26, -74.518, 126.137, -143.397, 38.209, 91.579, -80.857]
  MoveL 2208 to (-25.95, -54.63, 138.38) mm, rotated rx -155.44 ry 0 rz -25.68 deg; joints [21.291, -74.587, 126.218, -143.347, 38.209, 91.554, -80.88]
  MoveL 2209 to (-24.86, -55.33, 138.3) mm, rotated rx -155.45 ry 0 rz -25.46 deg; joints [21.306, -74.662, 126.279, -143.319, 38.21, 91.529, -81.099]
  MoveL 2210 to (-24.2, -56.01, 138.15) mm, rotated rx -155.3 ry 0 rz -24.6 deg; joints [21.286, -74.699, 126.269, -143.344, 38.21, 91.673, -81.904]
  MoveL 2211 to (-24.17, -55.99, 138.16) mm, rotated rx -155.58 ry 0 rz -21.61 deg; joints [21.255, -74.447, 126.093, -143.411, 38.21, 91.466, -84.947]
  MoveL 2212 to (-23.49, -55.66, 138.41) mm, rotated rx -155.82 ry 0 rz -21.1 deg; joints [21.286, -74.382, 126.105, -143.375, 38.211, 91.235, -85.541]
  MoveL 2213 to (-22.23, -55.42, 138.72) mm, rotated rx -155.82 ry 0 rz -21.1 deg; joints [21.32, -74.424, 126.175, -143.325, 38.211, 91.217, -85.579]
  MoveL 2214 to (-21.13, -55.63, 138.8) mm, rotated rx -155.84 ry 0 rz -20.91 deg; joints [21.342, -74.47, 126.231, -143.291, 38.211, 91.174, -85.786]
  MoveL 2215 to (-19.51, -56.28, 138.77) mm, rotated rx -155.82 ry 0 rz -19.22 deg; joints [21.338, -74.477, 126.23, -143.295, 38.211, 91.197, -87.461]
  MoveL 2216 to (-18.07, -56.32, 138.96) mm, rotated rx -156.03 ry 0 rz -17.2 deg; joints [21.353, -74.378, 126.203, -143.295, 38.224, 91.018, -89.542]
  MoveL 2217 to (-16.43, -56.97, 138.89) mm, rotated rx -156.03 ry 0 rz -17.2 deg; joints [21.381, -74.498, 126.305, -143.245, 38.224, 90.981, -89.538]
  MoveL 2218 to (-15.77, -57.73, 138.66) mm, rotated rx -156 ry 0 rz -17.05 deg; joints [21.38, -74.57, 126.341, -143.239, 38.224, 90.991, -89.649]
  MoveL 2219 to (-15.43, -58.46, 138.39) mm, rotated rx -155.45 ry 0 rz -14.9 deg; joints [21.29, -74.574, 126.213, -143.361, 38.224, 91.561, -91.656]
  MoveL 2220 to (-12.07, -59.39, 138.33) mm, rotated rx -155.39 ry 0 rz -11.63 deg; joints [21.283, -74.593, 126.212, -143.369, 38.224, 91.617, -94.896]
  MoveL 2221 to (-10.92, -60, 138.16) mm, rotated rx -155.39 ry 0 rz -11.63 deg; joints [21.297, -74.689, 126.283, -143.34, 38.224, 91.59, -94.88]
  MoveL 2222 to (-10.46, -60.5, 137.98) mm, rotated rx -155.37 ry 0 rz -11.57 deg; joints [21.295, -74.739, 126.306, -143.338, 38.224, 91.596, -94.925]
  MoveL 2223 to (-9.89, -61.32, 137.66) mm, rotated rx -155.07 ry 0 rz -10.87 deg; joints [21.254, -74.816, 126.288, -143.387, 38.224, 91.888, -95.524]
  MoveL 2224 to (-9.41, -61.94, 137.41) mm, rotated rx -155 ry 0 rz -10.6 deg; joints [21.241, -74.869, 126.293, -143.387, 38.207, 91.934, -95.759]
  MoveL 2225 to (-8.41, -64.13, 136.47) mm, rotated rx -154.15 ry 0 rz -9.35 deg; joints [21.122, -75.095, 126.25, -143.531, 38.207, 92.77, -96.73]
  MoveL 2226 to (-7.46, -65.27, 135.98) mm, rotated rx -153.57 ry 0 rz -8.1 deg; joints [21.042, -75.216, 126.208, -143.632, 38.207, 93.346, -97.806]
  MoveL 2227 to (-7.37, -65.37, 135.94) mm, rotated rx -153.23 ry 0 rz -6.19 deg; joints [20.974, -75.142, 126.075, -143.734, 38.207, 93.718, -99.639]
  MoveL 2228 to (-6.73, -65.37, 135.97) mm, rotated rx -153.26 ry 0 rz -5.63 deg; joints [20.979, -75.134, 126.076, -143.729, 38.207, 93.69, -100.205]
  MoveL 2229 to (-6.15, -65.42, 135.98) mm, rotated rx -153.26 ry 0 rz -5.38 deg; joints [20.984, -75.153, 126.094, -143.72, 38.207, 93.684, -100.453]
  MoveL 2230 to (-3.34, -65.88, 135.85) mm, rotated rx -153.16 ry 0 rz -3.13 deg; joints [20.972, -75.198, 126.098, -143.72, 38.189, 93.771, -102.688]
  MoveL 2231 to (-2.74, -66.04, 135.79) mm, rotated rx -153.16 ry 0 rz -3.13 deg; joints [20.979, -75.242, 126.132, -143.706, 38.189, 93.759, -102.683]
  MoveL 2232 to (-1.69, -66.7, 135.48) mm, rotated rx -152.83 ry 0 rz -1.4 deg; joints [20.92, -75.264, 126.066, -143.788, 38.189, 94.096, -104.304]
  MoveL 2233 to (-0.75, -66.76, 135.46) mm, rotated rx -152.84 ry 0 rz -1.09 deg; joints [20.929, -75.302, 126.1, -143.771, 38.189, 94.081, -104.618]
  MoveL 2234 to (-0.36, -66.92, 135.38) mm, rotated rx -152.95 ry 0 rz 1 deg; joints [20.901, -75.157, 125.982, -143.824, 38.189, 94.008, -106.718]
  MoveL 2235 to (0.64, -66.19, 135.74) mm, rotated rx -153.26 ry 0 rz 1.88 deg; joints [20.945, -75.073, 125.993, -143.769, 38.19, 93.703, -107.704]
  MoveL 2236 to (1.78, -65.71, 135.97) mm, rotated rx -153.26 ry 0 rz 1.88 deg; joints [20.976, -75.128, 126.065, -143.721, 38.19, 93.68, -107.73]
  MoveL 2237 to (2.93, -65.71, 135.95) mm, rotated rx -153.27 ry 0 rz 1.98 deg; joints [20.993, -75.196, 126.126, -143.69, 38.19, 93.652, -107.828]
  MoveL 2238 to (4, -65.92, 135.82) mm, rotated rx -153.16 ry 0 rz 2.9 deg; joints [20.977, -75.226, 126.121, -143.711, 38.19, 93.764, -108.711]
  MoveL 2239 to (7.3, -65.68, 135.79) mm, rotated rx -153.09 ry 0 rz 6.54 deg; joints [20.955, -75.183, 126.067, -143.746, 38.19, 93.848, -112.329]
  MoveL 2240 to (8.4, -65.81, 135.67) mm, rotated rx -153.09 ry 0 rz 6.54 deg; joints [20.968, -75.263, 126.129, -143.721, 38.19, 93.826, -112.318]
  MoveL 2241 to (9.29, -66.23, 135.4) mm, rotated rx -153.05 ry 0 rz 6.7 deg; joints [20.963, -75.334, 126.163, -143.721, 38.19, 93.849, -112.446]
  MoveL 2242 to (11.54, -67.79, 134.45) mm, rotated rx -152.22 ry 0 rz 8.46 deg; joints [20.843, -75.554, 126.129, -143.874, 38.19, 94.675, -113.935]
  MoveL 2243 to (12, -68.18, 134.21) mm, rotated rx -152.14 ry 0 rz 8.58 deg; joints [20.828, -75.604, 126.132, -143.874, 38.166, 94.731, -114.03]
  MoveL 2244 to (12.74, -68.99, 133.73) mm, rotated rx -151.8 ry 0 rz 8.99 deg; joints [20.776, -75.709, 126.126, -143.94, 38.166, 95.064, -114.326]
  MoveL 2245 to (13.57, -68.32, 134) mm, rotated rx -151.56 ry 0 rz 12.03 deg; joints [20.718, -75.55, 125.96, -144.037, 38.166, 95.367, -117.333]
  MoveL 2246 to (14.06, -68.11, 134.06) mm, rotated rx -151.6 ry 0 rz 12.47 deg; joints [20.725, -75.536, 125.961, -144.028, 38.166, 95.32, -117.792]
  MoveL 2247 to (18.3, -67.01, 134.08) mm, rotated rx -151.6 ry 0 rz 15.67 deg; joints [20.734, -75.566, 125.991, -144.013, 38.166, 95.315, -120.999]
  MoveL 2248 to (18.46, -66.21, 134.47) mm, rotated rx -151.82 ry 0 rz 16.26 deg; joints [20.768, -75.476, 125.991, -143.996, 38.2, 95.127, -121.644]
  MoveL 2249 to (19.9, -64.86, 134.93) mm, rotated rx -152.3 ry 0 rz 17.63 deg; joints [20.836, -75.363, 126.014, -143.907, 38.2, 94.642, -123.157]
  MoveL 2250 to (20.58, -64.61, 134.95) mm, rotated rx -152.32 ry 0 rz 18.25 deg; joints [20.838, -75.358, 126.014, -143.905, 38.201, 94.628, -123.784]
  MoveL 2251 to (26.87, -62.57, 134.8) mm, rotated rx -152.17 ry 0 rz 23.69 deg; joints [20.82, -75.406, 126.014, -143.917, 38.187, 94.76, -129.19]
  MoveL 2252 to (28.7, -61.62, 134.86) mm, rotated rx -152.22 ry 0 rz 25.68 deg; joints [20.822, -75.372, 125.997, -143.917, 38.187, 94.721, -131.196]
  MoveL 2253 to (29.82, -61.29, 134.76) mm, rotated rx -152.22 ry 0 rz 25.68 deg; joints [20.837, -75.455, 126.065, -143.888, 38.187, 94.697, -131.188]
  MoveL 2254 to (30.96, -61.36, 134.47) mm, rotated rx -152.17 ry 0 rz 25.88 deg; joints [20.833, -75.536, 126.106, -143.888, 38.187, 94.722, -131.35]
  MoveL 2255 to (32.73, -61.9, 133.81) mm, rotated rx -151.32 ry 0 rz 28.15 deg; joints [20.699, -75.647, 125.998, -144.072, 38.187, 95.599, -133.376]
  MoveL 2256 to (34.2, -61.35, 133.7) mm, rotated rx -151.22 ry 0 rz 29.45 deg; joints [20.684, -75.672, 125.993, -144.092, 38.187, 95.702, -134.644]
  MoveL 2257 to (34.89, -61.18, 133.6) mm, rotated rx -151.2 ry 0 rz 29.59 deg; joints [20.686, -75.718, 126.022, -144.085, 38.187, 95.717, -134.764]
  MoveL 2258 to (35.94, -61.16, 133.33) mm, rotated rx -150.91 ry 0 rz 31.34 deg; joints [20.624, -75.71, 125.941, -144.175, 38.187, 96.035, -136.43]
  MoveL 2259 to (37.28, -60.11, 133.44) mm, rotated rx -150.99 ry 0 rz 32.74 deg; joints [20.637, -75.684, 125.941, -144.159, 38.187, 95.95, -137.854]
  MoveL 2260 to (37.77, -59.72, 133.48) mm, rotated rx -151.02 ry 0 rz 33.23 deg; joints [20.642, -75.678, 125.943, -144.152, 38.187, 95.923, -138.351]
  MoveL 2261 to (38.36, -59.36, 133.47) mm, rotated rx -151.02 ry 0 rz 33.23 deg; joints [20.653, -75.723, 125.984, -144.132, 38.187, 95.909, -138.352]
  MoveL 2262 to (43.48, -56.74, 133.04) mm, rotated rx -150.64 ry 0 rz 37.88 deg; joints [20.596, -75.819, 125.97, -144.208, 38.187, 96.291, -142.883]
  MoveL 2263 to (44.61, -56.39, 132.8) mm, rotated rx -150.64 ry 0 rz 37.88 deg; joints [20.605, -75.91, 126.034, -144.189, 38.187, 96.269, -142.863]
  MoveL 2264 to (45.13, -56.35, 132.64) mm, rotated rx -150.55 ry 0 rz 38.11 deg; joints [20.59, -75.947, 126.034, -144.195, 38.171, 96.343, -143.076]
  MoveL 2265 to (47.13, -56.37, 131.95) mm, rotated rx -149.73 ry 0 rz 40.67 deg; joints [20.45, -76.036, 125.916, -144.393, 38.171, 97.204, -145.392]
  MoveL 2266 to (50.68, -53.13, 131.95) mm, rotated rx -150.39 ry 0 rz 43.42 deg; joints [20.536, -76.002, 126.001, -144.27, 38.171, 96.515, -148.283]
  MoveL 2267 to (51.14, -52.77, 131.92) mm, rotated rx -150.38 ry 0 rz 43.51 deg; joints [20.542, -76.036, 126.028, -144.259, 38.171, 96.514, -148.375]
  MoveL 2268 to (52.56, -50.63, 132.2) mm, rotated rx -150.61 ry 0 rz 45.52 deg; joints [20.575, -75.97, 126.03, -144.215, 38.171, 96.285, -150.454]
  MoveL 2269 to (59.81, -57.33, 149.59) mm, rotated rx -150.59 ry 0 rz 45.74 deg; joints [21.451, -75.971, 125.891, -143.955, 39.973, 96.285, -148.948]
  Set speed (1000.0 mm/s)
  MoveL 2270 to (61.99, -54.39, 149.8) mm, rotated rx -150.73 ry 0 rz 48.5 deg; joints [21.469, -75.906, 125.883, -143.955, 40.004, 96.172, -151.737]
  Set speed (5.0 mm/s)
  MoveL 2271 to (54.66, -47.91, 132.36) mm, rotated rx -150.73 ry 0 rz 48.5 deg; joints [20.588, -75.913, 126.011, -144.201, 38.17, 96.172, -153.476]
  Set speed (16.7 mm/s)
  MoveL 2272 to (55.79, -46.79, 132.29) mm, rotated rx -150.67 ry 0 rz 49.8 deg; joints [20.578, -75.924, 126.006, -144.214, 38.17, 96.229, -154.753]
  MoveL 2273 to (56.07, -46.15, 132.39) mm, rotated rx -150.78 ry 0 rz 50.94 deg; joints [20.579, -75.847, 125.962, -144.218, 38.17, 96.141, -155.93]
  MoveL 2274 to (56.83, -45.24, 132.38) mm, rotated rx -150.78 ry 0 rz 50.94 deg; joints [20.599, -75.925, 126.032, -144.183, 38.17, 96.117, -155.932]
  MoveL 2275 to (57.77, -44.66, 132.18) mm, rotated rx -150.75 ry 0 rz 51.17 deg; joints [20.6, -75.995, 126.075, -144.176, 38.17, 96.131, -156.136]
  MoveL 2276 to (60.3, -43.63, 131.38) mm, rotated rx -150.12 ry 0 rz 53.08 deg; joints [20.502, -76.163, 126.056, -144.308, 38.17, 96.77, -157.844]
  MoveL 2277 to (61.86, -41.57, 131.32) mm, rotated rx -149.91 ry 0 rz 56.12 deg; joints [20.456, -76.116, 125.972, -144.379, 38.17, 97.01, -160.824]
  MoveL 2278 to (62.57, -39.87, 131.52) mm, rotated rx -150.07 ry 0 rz 58 deg; joints [20.471, -76.033, 125.946, -144.379, 38.192, 96.875, -162.737]
  MoveL 2279 to (63.23, -38.94, 131.48) mm, rotated rx -150.07 ry 0 rz 58 deg; joints [20.489, -76.11, 126.013, -144.348, 38.192, 96.851, -162.736]
  MoveL 2280 to (63.85, -38.47, 131.32) mm, rotated rx -150.05 ry 0 rz 58.09 deg; joints [20.491, -76.164, 126.048, -144.341, 38.192, 96.853, -162.812]
  MoveL 2281 to (64.49, -38.1, 131.11) mm, rotated rx -149.89 ry 0 rz 58.61 deg; joints [20.465, -76.208, 126.043, -144.376, 38.192, 97.021, -163.28]
  MoveL 2282 to (64.68, -37.79, 131.11) mm, rotated rx -149.74 ry 0 rz 59.75 deg; joints [20.431, -76.161, 125.975, -144.429, 38.192, 97.194, -164.389]
  MoveL 2283 to (65.32, -37.14, 130.98) mm, rotated rx -149.74 ry 0 rz 59.75 deg; joints [20.441, -76.229, 126.03, -144.417, 38.202, 97.183, -164.37]
  MoveL 2284 to (65.81, -36.84, 130.82) mm, rotated rx -149.72 ry 0 rz 59.82 deg; joints [20.439, -76.271, 126.054, -144.417, 38.202, 97.194, -164.422]
  MoveL 2285 to (66.52, -36.5, 130.55) mm, rotated rx -149.51 ry 0 rz 60.34 deg; joints [20.406, -76.327, 126.049, -144.462, 38.202, 97.406, -164.868]
  MoveL 2286 to (70.08, -32.64, 129.71) mm, rotated rx -148.7 ry 0 rz 64.84 deg; joints [20.271, -76.476, 125.982, -144.652, 38.202, 98.259, -169.125]
  MoveL 2287 to (70.59, -32.15, 129.55) mm, rotated rx -148.63 ry 0 rz 65.08 deg; joints [20.262, -76.52, 125.996, -144.652, 38.189, 98.31, -169.351]
  MoveL 2288 to (72.16, -30.71, 129.03) mm, rotated rx -148.24 ry 0 rz 66.57 deg; joints [20.198, -76.625, 125.988, -144.741, 38.189, 98.714, -170.715]
  MoveL 2289 to (72.5, -29.55, 129.13) mm, rotated rx -148.2 ry 0 rz 68.17 deg; joints [20.181, -76.563, 125.929, -144.77, 38.189, 98.777, -172.313]
  MoveL 2290 to (72.86, -28.78, 129.09) mm, rotated rx -148.17 ry 0 rz 68.81 deg; joints [20.177, -76.569, 125.928, -144.777, 38.189, 98.805, -172.941]
  MoveL 2291 to (73.21, -28.21, 129.02) mm, rotated rx -148.17 ry 0 rz 68.81 deg; joints [20.185, -76.617, 125.967, -144.762, 38.189, 98.792, -172.936]
  MoveL 2292 to (79.18, -19.42, 127.09) mm, rotated rx -146.78 ry 0 rz 76.24 deg; joints [19.952, -76.999, 125.951, -145.09, 38.189, 100.241, -179.92]
  MoveL 2293 to (84.02, -9.55, 125.11) mm, rotated rx -145.33 ry 0 rz 83.75 deg; joints [20.327, -77.597, 129.279, -150.007, 47.579, 106.369, -180]
  MoveL 2294 to (85.47, -8.13, 124.22) mm, rotated rx -145.33 ry 0 rz 83.75 deg; joints [20.317, -77.765, 129.388, -150.018, 47.579, 106.353, -179.942]
  MoveL 2295 to (86.56, -8.17, 123.47) mm, rotated rx -145.33 ry 0 rz 83.75 deg; joints [20.285, -77.833, 129.399, -150.054, 47.57, 106.353, -179.89]
  MoveL 2296 to (87.6, -9.12, 122.67) mm, rotated rx -145.33 ry 0 rz 83.75 deg; joints [20.237, -77.849, 129.359, -150.119, 47.57, 106.369, -179.822]
  MoveL 2297 to (87.88, -11, 122.34) mm, rotated rx -145.33 ry 0 rz 83.75 deg; joints [20.19, -77.766, 129.249, -150.183, 47.57, 106.397, -179.783]
  MoveL 2298 to (85.96, -19.02, 122.71) mm, rotated rx -145.61 ry 0 rz 78.27 deg; joints [20.239, -77.692, 129.249, -150.119, 47.571, 106.113, -174.391]
  MoveL 2299 to (82.72, -28.28, 123.17) mm, rotated rx -145.94 ry 0 rz 71.71 deg; joints [20.297, -77.603, 129.248, -150.043, 47.571, 105.772, -167.925]
  MoveL 2300 to (79.9, -32.89, 123.88) mm, rotated rx -146.4 ry 0 rz 68.39 deg; joints [20.372, -77.431, 129.207, -149.947, 47.572, 105.298, -164.755]
  MoveL 2301 to (79.79, -32.88, 123.91) mm, rotated rx -144.76 ry 0 rz 66.87 deg; joints [20.213, -77.905, 129.256, -149.947, 47.138, 106.763, -163.247]
  MoveL 2302 to (81.28, -31.88, 123.21) mm, rotated rx -144.28 ry 0 rz 67.89 deg; joints [20.129, -78.06, 129.279, -150.056, 47.138, 107.26, -164.126]
  MoveL 2303 to (83.27, -31.68, 121.93) mm, rotated rx -144.25 ry 0 rz 67.84 deg; joints [20.086, -78.231, 129.341, -150.084, 47.08, 107.26, -164.017]
  MoveL 2304 to (84.18, -32.65, 121.06) mm, rotated rx -144.23 ry 0 rz 67.8 deg; joints [20.038, -78.274, 129.323, -150.148, 47.08, 107.292, -163.907]
  MoveL 2305 to (84.06, -35.02, 120.5) mm, rotated rx -144.21 ry 0 rz 67.74 deg; joints [19.974, -78.197, 129.199, -150.238, 47.08, 107.355, -163.785]
  MoveL 2306 to (83.49, -36.19, 120.53) mm, rotated rx -144.05 ry 0 rz 65.89 deg; joints [19.986, -78.326, 129.306, -150.219, 47.08, 107.498, -161.918]
  MoveL 2307 to (83.76, -38.69, 119.57) mm, rotated rx -143.44 ry 0 rz 64.52 deg; joints [19.871, -78.528, 129.306, -150.317, 46.965, 108.082, -160.441]
  MoveL 2308 to (85.01, -41.41, 117.75) mm, rotated rx -142.04 ry 0 rz 63 deg; joints [19.623, -78.989, 129.306, -150.485, 46.62, 109.4, -158.782]
  MoveL 2309 to (84.94, -43.5, 117.06) mm, rotated rx -142.04 ry 0 rz 63 deg; joints [19.561, -78.927, 129.199, -150.572, 46.62, 109.436, -158.72]
  MoveL 2310 to (84.41, -44.47, 117.08) mm, rotated rx -142.03 ry 0 rz 62.8 deg; joints [19.547, -78.881, 129.152, -150.591, 46.62, 109.457, -158.518]
  MoveL 2311 to (82.72, -46.56, 117.46) mm, rotated rx -142.26 ry 0 rz 61.22 deg; joints [19.593, -78.804, 129.152, -150.551, 46.665, 109.23, -156.97]
  MoveL 2312 to (82.46, -48.44, 116.89) mm, rotated rx -141.93 ry 0 rz 59.57 deg; joints [19.537, -78.973, 129.179, -150.551, 46.509, 109.506, -155.34]
  MoveL 2313 to (82.16, -49.29, 116.74) mm, rotated rx -141.81 ry 0 rz 58.79 deg; joints [19.521, -79.032, 129.197, -150.551, 46.466, 109.606, -154.565]
  MoveL 2314 to (82.94, -48.44, 116.52) mm, rotated rx -139.92 ry 0 rz 59.15 deg; joints [19.275, -79.463, 129.197, -150.724, 46.131, 111.433, -154.794]
  MoveL 2315 to (83.88, -47.94, 116.06) mm, rotated rx -139.87 ry 0 rz 59.29 deg; joints [19.258, -79.548, 129.231, -150.724, 46.082, 111.465, -154.934]
  MoveL 2316 to (86.1, -47.26, 114.71) mm, rotated rx -139.06 ry 0 rz 60.28 deg; joints [19.089, -79.809, 129.231, -150.874, 45.914, 112.267, -155.806]
  MoveL 2317 to (87.26, -46.57, 114.11) mm, rotated rx -138.59 ry 0 rz 61.13 deg; joints [18.998, -79.929, 129.231, -150.982, 45.876, 112.756, -156.56]
  MoveL 2318 to (88.1, -46.23, 113.6) mm, rotated rx -138.26 ry 0 rz 61.22 deg; joints [18.933, -80.063, 129.231, -150.994, 45.716, 113.047, -156.667]
  MoveL 2319 to (89.65, -47.03, 112.04) mm, rotated rx -137.49 ry 0 rz 61.4 deg; joints [18.755, -80.308, 129.231, -151.18, 45.587, 113.836, -156.704]
  MoveL 2320 to (90.94, -46.5, 111.23) mm, rotated rx -137.02 ry 0 rz 62.03 deg; joints [18.652, -80.455, 129.231, -151.276, 45.49, 114.314, -157.261]
  MoveL 2321 to (92.41, -46.56, 109.99) mm, rotated rx -137.02 ry 0 rz 62.03 deg; joints [18.606, -80.578, 129.278, -151.321, 45.451, 114.314, -157.216]
  MoveL 2322 to (104.65, -53.08, 124.41) mm, rotated rx -136.91 ry 0 rz 62.02 deg; joints [19.362, -80.94, 129.04, -150.597, 46.317, 113.784, -155.995]
  Set speed (1000.0 mm/s)
  MoveL 2323 to (106.64, -54.76, 121.97) mm, rotated rx -135.66 ry 0 rz 61.75 deg; joints [19.074, -81.355, 129.04, -150.842, 45.992, 115.033, -155.584]
  Set speed (5.0 mm/s)
  MoveL 2324 to (94.32, -48.14, 107.66) mm, rotated rx -135.66 ry 0 rz 61.75 deg; joints [18.363, -81.034, 129.601, -151.922, 45.992, 116.019, -156.162]
  Set speed (16.7 mm/s)
  MoveL 2325 to (94.76, -48.45, 107.15) mm, rotated rx -135.6 ry 0 rz 61.75 deg; joints [18.329, -81.077, 129.601, -151.958, 45.967, 116.093, -156.138]
  MoveL 2326 to (95.38, -49.1, 106.29) mm, rotated rx -135.13 ry 0 rz 61.6 deg; joints [18.222, -81.224, 129.601, -152.055, 45.853, 116.565, -155.935]
  MoveL 2327 to (96.58, -49.18, 105.16) mm, rotated rx -134.03 ry 0 rz 61.88 deg; joints [18.007, -81.509, 129.602, -152.255, 45.633, 117.689, -156.111]
  MoveL 2328 to (97.3, -49.5, 104.35) mm, rotated rx -134.03 ry 0 rz 61.88 deg; joints [17.969, -81.563, 129.602, -152.285, 45.585, 117.689, -156.1]
  MoveL 2329 to (97.87, -50.47, 103.35) mm, rotated rx -133.95 ry 0 rz 61.86 deg; joints [17.906, -81.61, 129.592, -152.376, 45.585, 117.808, -156.007]
  MoveL 2330 to (98.14, -51.93, 102.37) mm, rotated rx -133.43 ry 0 rz 61.25 deg; joints [17.782, -81.771, 129.592, -152.489, 45.452, 118.338, -155.351]
  MoveL 2331 to (97.89, -53.62, 101.74) mm, rotated rx -133.43 ry 0 rz 61.25 deg; joints [17.729, -81.712, 129.504, -152.566, 45.452, 118.378, -155.306]
  MoveL 2332 to (96.76, -55.02, 102.08) mm, rotated rx -133.43 ry 0 rz 61.25 deg; joints [17.715, -81.581, 129.388, -152.587, 45.452, 118.396, -155.315]
  MoveL 2333 to (96.07, -55.49, 102.48) mm, rotated rx -133.64 ry 0 rz 60.86 deg; joints [17.765, -81.517, 129.387, -152.54, 45.504, 118.177, -154.948]
  MoveL 2334 to (88.95, -59.16, 106.76) mm, rotated rx -135.86 ry 0 rz 57.36 deg; joints [18.289, -80.808, 129.387, -152.072, 46.08, 115.921, -151.669]
  MoveL 2335 to (88.14, -59.55, 107.21) mm, rotated rx -136.12 ry 0 rz 56.94 deg; joints [18.347, -80.728, 129.387, -152.018, 46.14, 115.655, -151.277]
  MoveL 2336 to (87.61, -59.73, 107.55) mm, rotated rx -136.12 ry 0 rz 56.94 deg; joints [18.355, -80.679, 129.355, -152.009, 46.142, 115.655, -151.293]
  MoveL 2337 to (78.4, -60.94, 113.79) mm, rotated rx -139.66 ry 0 rz 53.39 deg; joints [19.125, -79.546, 129.352, -151.313, 46.933, 112.113, -148.208]
  MoveL 2338 to (77.11, -60.45, 114.92) mm, rotated rx -139.66 ry 0 rz 53.39 deg; joints [19.169, -79.441, 129.321, -151.268, 46.965, 112.113, -148.256]
  MoveL 2339 to (76.61, -59.54, 115.72) mm, rotated rx -139.74 ry 0 rz 53.41 deg; joints [19.221, -79.389, 129.328, -151.198, 46.965, 112.008, -148.347]
  MoveL 2340 to (76.35, -58.13, 116.62) mm, rotated rx -140.9 ry 0 rz 54.26 deg; joints [19.408, -79.057, 129.328, -151.073, 47.242, 110.897, -149.28]
  MoveL 2341 to (75.78, -57.8, 117.15) mm, rotated rx -141.23 ry 0 rz 54.22 deg; joints [19.474, -78.95, 129.328, -151.016, 47.31, 110.577, -149.285]
  MoveL 2342 to (75.2, -57.32, 117.75) mm, rotated rx -141.42 ry 0 rz 54.25 deg; joints [19.525, -78.865, 129.328, -150.971, 47.362, 110.393, -149.358]
  MoveL 2343 to (74.91, -56.95, 118.12) mm, rotated rx -141.48 ry 0 rz 54.28 deg; joints [19.55, -78.83, 129.328, -150.942, 47.371, 110.329, -149.416]
  MoveL 2344 to (73.34, -58.83, 118.2) mm, rotated rx -142.66 ry 0 rz 51.91 deg; joints [19.713, -78.668, 129.364, -150.722, 47.371, 109.093, -147.285]
  MoveL 2345 to (70.71, -60.37, 119) mm, rotated rx -143.17 ry 0 rz 50.14 deg; joints [19.805, -78.501, 129.333, -150.599, 47.372, 108.56, -145.667]
  MoveL 2346 to (70.79, -60.67, 118.79) mm, rotated rx -141.63 ry 0 rz 48.04 deg; joints [19.65, -79.027, 129.45, -150.599, 46.939, 109.927, -143.597]
  MoveL 2347 to (71.84, -60.7, 118.15) mm, rotated rx -141.23 ry 0 rz 48.48 deg; joints [19.57, -79.158, 129.451, -150.672, 46.865, 110.325, -143.962]
  MoveL 2348 to (73.06, -61.14, 117.19) mm, rotated rx -141.2 ry 0 rz 48.45 deg; joints [19.529, -79.266, 129.469, -150.687, 46.779, 110.325, -143.934]
  MoveL 2349 to (73.58, -62.13, 116.35) mm, rotated rx -141.18 ry 0 rz 48.44 deg; joints [19.483, -79.313, 129.461, -150.749, 46.779, 110.366, -143.851]
  MoveL 2350 to (73.11, -64.05, 115.6) mm, rotated rx -141.14 ry 0 rz 48.41 deg; joints [19.418, -79.274, 129.369, -150.84, 46.779, 110.439, -143.753]
  MoveL 2351 to (71.05, -67.17, 115.11) mm, rotated rx -140.85 ry 0 rz 46.19 deg; joints [19.359, -79.375, 129.369, -150.884, 46.703, 110.721, -141.497]
  MoveL 2352 to (70.39, -67.87, 115.11) mm, rotated rx -140.85 ry 0 rz 46.19 deg; joints [19.342, -79.317, 129.31, -150.908, 46.703, 110.735, -141.49]
  MoveL 2353 to (69.96, -68.2, 115.17) mm, rotated rx -140.88 ry 0 rz 45.86 deg; joints [19.349, -79.306, 129.309, -150.9, 46.707, 110.697, -141.177]
  MoveL 2354 to (66.65, -69.89, 116.11) mm, rotated rx -141.38 ry 0 rz 44.07 deg; joints [19.452, -79.105, 129.307, -150.849, 46.894, 110.245, -139.407]
  MoveL 2355 to (66.68, -69.85, 116.12) mm, rotated rx -141.37 ry 0 rz 42.8 deg; joints [19.489, -79.24, 129.444, -150.796, 46.894, 110.228, -138.143]
  MoveL 2356 to (66.19, -70.87, 115.79) mm, rotated rx -141.17 ry 0 rz 42.16 deg; joints [19.449, -79.307, 129.444, -150.83, 46.85, 110.424, -137.476]
  MoveL 2357 to (65.72, -71.55, 115.64) mm, rotated rx -141.17 ry 0 rz 42.16 deg; joints [19.428, -79.27, 129.396, -150.859, 46.85, 110.438, -137.46]
  MoveL 2358 to (64.95, -72.39, 115.55) mm, rotated rx -141.11 ry 0 rz 41.47 deg; joints [19.417, -79.29, 129.396, -150.866, 46.833, 110.49, -136.772]
  MoveL 2359 to (60.06, -77.65, 114.76) mm, rotated rx -140.63 ry 0 rz 37.13 deg; joints [19.321, -79.462, 129.396, -150.926, 46.683, 110.941, -132.398]
  MoveL 2360 to (60, -77.7, 114.78) mm, rotated rx -139.79 ry 0 rz 35.86 deg; joints [19.243, -79.756, 129.487, -150.926, 46.466, 111.695, -131.138]
  MoveL 2361 to (60.17, -78.25, 114.31) mm, rotated rx -139.7 ry 0 rz 35.81 deg; joints [19.209, -79.802, 129.487, -150.964, 46.449, 111.793, -131.056]
  MoveL 2362 to (60.29, -79.98, 113.05) mm, rotated rx -139.09 ry 0 rz 35.35 deg; joints [19.07, -80.009, 129.487, -151.099, 46.329, 112.407, -130.488]
  MoveL 2363 to (60.74, -80.98, 112.08) mm, rotated rx -138.27 ry 0 rz 35.1 deg; joints [18.917, -80.254, 129.487, -151.216, 46.133, 113.206, -130.169]
  MoveL 2364 to (61.07, -81.61, 111.43) mm, rotated rx -136.88 ry 0 rz 35.79 deg; joints [18.689, -80.506, 129.487, -151.53, 46.123, 114.704, -130.556]
  MoveL 2365 to (63.9, -80.82, 110.4) mm, rotated rx -136.3 ry 0 rz 37.36 deg; joints [18.559, -80.686, 129.487, -151.652, 46.001, 115.291, -132.049]
  MoveL 2366 to (63.79, -80.87, 110.43) mm, rotated rx -136.29 ry 0 rz 38.55 deg; joints [18.521, -80.55, 129.347, -151.708, 46.001, 115.337, -133.225]
  MoveL 2367 to (64.44, -79.87, 110.78) mm, rotated rx -136.49 ry 0 rz 39.2 deg; joints [18.566, -80.484, 129.347, -151.669, 46.053, 115.135, -133.892]
  MoveL 2368 to (65.17, -79.06, 110.94) mm, rotated rx -136.49 ry 0 rz 39.2 deg; joints [18.591, -80.539, 129.411, -151.634, 46.053, 115.116, -133.908]
  MoveL 2369 to (66.37, -78.32, 110.76) mm, rotated rx -136.49 ry 0 rz 39.39 deg; joints [18.6, -80.617, 129.481, -151.62, 46.053, 115.107, -134.09]
  MoveL 2370 to (68.83, -77.4, 109.9) mm, rotated rx -136.01 ry 0 rz 40.79 deg; joints [18.492, -80.767, 129.481, -151.723, 45.951, 115.598, -135.429]
  MoveL 2371 to (70.19, -76.87, 109.4) mm, rotated rx -135.73 ry 0 rz 41.57 deg; joints [18.429, -80.854, 129.481, -151.782, 45.889, 115.88, -136.168]
  MoveL 2372 to (70.42, -76.02, 109.85) mm, rotated rx -135.82 ry 0 rz 42.09 deg; joints [18.461, -80.794, 129.478, -151.767, 45.952, 115.804, -136.689]
  MoveL 2373 to (71.95, -74.45, 109.94) mm, rotated rx -136.01 ry 0 rz 43.29 deg; joints [18.493, -80.752, 129.478, -151.736, 45.979, 115.607, -137.905]
  MoveL 2374 to (72.52, -74.17, 109.75) mm, rotated rx -135.91 ry 0 rz 43.63 deg; joints [18.469, -80.784, 129.478, -151.758, 45.958, 115.712, -138.232]
  MoveL 2375 to (73.43, -73.9, 109.33) mm, rotated rx -135.91 ry 0 rz 43.63 deg; joints [18.465, -80.864, 129.538, -151.763, 45.958, 115.709, -138.212]
  MoveL 2376 to (79.17, -73.12, 105.8) mm, rotated rx -133.95 ry 0 rz 46.2 deg; joints [18.014, -81.47, 129.538, -152.185, 45.509, 117.71, -140.543]
  MoveL 2377 to (82.04, -72.14, 104.27) mm, rotated rx -133.03 ry 0 rz 47.79 deg; joints [17.802, -81.726, 129.538, -152.409, 45.344, 118.683, -142.003]
  MoveL 2378 to (82.67, -71.97, 103.89) mm, rotated rx -132.95 ry 0 rz 47.91 deg; joints [17.775, -81.781, 129.539, -152.409, 45.263, 118.738, -142.14]
  MoveL 2379 to (85.46, -71.42, 102) mm, rotated rx -131.86 ry 0 rz 49.15 deg; joints [17.517, -82.098, 129.539, -152.662, 45.019, 119.884, -143.264]
  MoveL 2380 to (86.69, -71.65, 100.79) mm, rotated rx -131.86 ry 0 rz 49.15 deg; joints [17.469, -82.207, 129.577, -152.701, 44.958, 119.884, -143.246]
  MoveL 2381 to (87.19, -72.43, 99.79) mm, rotated rx -131.79 ry 0 rz 49.15 deg; joints [17.409, -82.266, 129.577, -152.778, 44.938, 119.986, -143.194]
  MoveL 2382 to (87.39, -73.34, 98.95) mm, rotated rx -131.37 ry 0 rz 48.87 deg; joints [17.304, -82.393, 129.577, -152.878, 44.829, 120.427, -142.874]
  MoveL 2383 to (88.05, -74.11, 97.79) mm, rotated rx -130.47 ry 0 rz 48.68 deg; joints [17.109, -82.639, 129.577, -153.046, 44.589, 121.341, -142.634]
  MoveL 2384 to (99.47, -84.16, 110.77) mm, rotated rx -130.47 ry 0 rz 48.68 deg; joints [17.777, -83.062, 129.067, -152.009, 44.59, 120.359, -141.984]
  Set speed (1000.0 mm/s)
  MoveL 2385 to (96.52, -88.4, 110.08) mm, rotated rx -130.58 ry 0 rz 48.38 deg; joints [17.691, -82.807, 128.8, -152.138, 44.592, 120.331, -141.64]
  Set speed (5.0 mm/s)
  MoveL 2386 to (85.16, -78.31, 97.07) mm, rotated rx -130.58 ry 0 rz 48.38 deg; joints [17.024, -82.384, 129.308, -153.174, 44.592, 121.311, -142.291]
  Set speed (16.7 mm/s)
  MoveL 2387 to (84.42, -78.42, 97.62) mm, rotated rx -130.86 ry 0 rz 48.09 deg; joints [17.093, -82.302, 129.308, -153.107, 44.663, 121.022, -142.035]
  MoveL 2388 to (84.43, -78.36, 97.65) mm, rotated rx -130.44 ry 0 rz 45.91 deg; joints [17.103, -82.658, 129.611, -153.09, 44.663, 121.411, -139.8]
  MoveL 2389 to (85.4, -79.89, 95.56) mm, rotated rx -129.41 ry 0 rz 45.7 deg; joints [16.837, -82.965, 129.611, -153.348, 44.391, 122.505, -139.502]
  MoveL 2390 to (86.47, -80.7, 93.9) mm, rotated rx -128.4 ry 0 rz 45.76 deg; joints [16.593, -83.24, 129.611, -153.586, 44.139, 123.578, -139.498]
  MoveL 2391 to (86.78, -81.13, 93.24) mm, rotated rx -128.3 ry 0 rz 45.74 deg; joints [16.545, -83.29, 129.611, -153.636, 44.097, 123.689, -139.457]
  MoveL 2392 to (87.3, -83.14, 90.96) mm, rotated rx -127.39 ry 0 rz 45.29 deg; joints [16.281, -83.567, 129.611, -153.91, 43.853, 124.696, -138.915]
  MoveL 2393 to (87.98, -84.68, 88.86) mm, rotated rx -126.27 ry 0 rz 44.95 deg; joints [15.991, -83.874, 129.611, -154.196, 43.549, 125.902, -138.515]
  MoveL 2394 to (88.07, -85.09, 88.38) mm, rotated rx -126.27 ry 0 rz 44.95 deg; joints [15.965, -83.886, 129.607, -154.234, 43.549, 125.922, -138.492]
  MoveL 2395 to (87.89, -86.33, 87.35) mm, rotated rx -126.12 ry 0 rz 44.86 deg; joints [15.883, -83.919, 129.588, -154.357, 43.548, 126.135, -138.321]
  MoveL 2396 to (86.28, -89.88, 85.35) mm, rotated rx -125.37 ry 0 rz 43.46 deg; joints [15.653, -84.114, 129.588, -154.638, 43.417, 127.01, -136.809]
  MoveL 2397 to (85.37, -91.08, 85.01) mm, rotated rx -125.37 ry 0 rz 43.46 deg; joints [15.616, -84.038, 129.502, -154.694, 43.417, 127.045, -136.787]
  MoveL 2398 to (84.57, -91.73, 85.12) mm, rotated rx -125.38 ry 0 rz 43.3 deg; joints [15.612, -83.989, 129.457, -154.701, 43.417, 127.046, -136.629]
  MoveL 2399 to (83.35, -92.49, 85.48) mm, rotated rx -125.55 ry 0 rz 42.64 deg; joints [15.66, -83.942, 129.457, -154.649, 43.461, 126.851, -135.982]
  MoveL 2400 to (83.33, -92.48, 85.48) mm, rotated rx -125.31 ry 0 rz 41.43 deg; joints [15.658, -84.153, 129.638, -154.649, 43.457, 127.09, -134.747]
  MoveL 2401 to (82.96, -93.63, 84.59) mm, rotated rx -124.89 ry 0 rz 40.95 deg; joints [15.543, -84.267, 129.638, -154.769, 43.343, 127.547, -134.244]
  MoveL 2402 to (82.93, -93.6, 84.67) mm, rotated rx -124.13 ry 0 rz 40.24 deg; joints [15.42, -84.468, 129.638, -154.787, 42.993, 128.256, -133.671]
  MoveL 2403 to (83.7, -94.23, 83.21) mm, rotated rx -123.45 ry 0 rz 40.33 deg; joints [15.227, -84.648, 129.638, -154.991, 42.81, 129.018, -133.72]
  MoveL 2404 to (84.01, -94.85, 82.19) mm, rotated rx -123.45 ry 0 rz 40.33 deg; joints [15.176, -84.687, 129.638, -155.058, 42.788, 129.052, -133.691]
  MoveL 2405 to (83.95, -95.66, 81.3) mm, rotated rx -123.29 ry 0 rz 40.25 deg; joints [15.102, -84.734, 129.638, -155.165, 42.775, 129.27, -133.557]
  MoveL 2406 to (83.68, -96.53, 80.53) mm, rotated rx -122.97 ry 0 rz 39.94 deg; joints [15.006, -84.818, 129.638, -155.272, 42.693, 129.64, -133.216]
  MoveL 2407 to (83.66, -96.49, 80.59) mm, rotated rx -121.55 ry 0 rz 40.21 deg; joints [14.748, -85.016, 129.638, -155.592, 42.54, 131.216, -133.379]
  MoveL 2408 to (84.44, -96.18, 80.17) mm, rotated rx -121.35 ry 0 rz 40.58 deg; joints [14.691, -85.065, 129.638, -155.656, 42.489, 131.441, -133.735]
  MoveL 2409 to (84.87, -96, 79.93) mm, rotated rx -121.24 ry 0 rz 40.77 deg; joints [14.659, -85.093, 129.638, -155.69, 42.46, 131.564, -133.928]
  MoveL 2410 to (89.89, -94.29, 76.4) mm, rotated rx -119.67 ry 0 rz 42.92 deg; joints [14.19, -85.491, 129.638, -156.207, 42.025, 133.38, -136.007]
  MoveL 2411 to (90.53, -94.13, 75.84) mm, rotated rx -119.54 ry 0 rz 43.04 deg; joints [14.141, -85.547, 129.638, -156.241, 41.935, 133.509, -136.15]
  MoveL 2412 to (91.88, -94.11, 74.2) mm, rotated rx -119.02 ry 0 rz 43.33 deg; joints [13.96, -85.707, 129.638, -156.423, 41.727, 134.113, -136.454]
  MoveL 2413 to (85.22, -103.24, 69.89) mm, rotated rx -117.88 ry 0 rz 40.55 deg; joints [13.491, -85.794, 129.52, -157.151, 41.727, 135.701, -133.333]
  MoveL 2414 to (84.46, -103.07, 71.07) mm, rotated rx -118.39 ry 0 rz 40.35 deg; joints [13.647, -85.675, 129.52, -156.972, 41.865, 135.105, -133.15]
  MoveL 2415 to (82.9, -103.3, 72.55) mm, rotated rx -119.34 ry 0 rz 39.47 deg; joints [13.906, -85.507, 129.52, -156.633, 41.996, 133.96, -132.375]
  MoveL 2416 to (82.42, -103.29, 73.11) mm, rotated rx -119.4 ry 0 rz 39.44 deg; joints [13.942, -85.463, 129.52, -156.61, 42.072, 133.903, -132.321]
  MoveL 2417 to (81.9, -103.11, 73.93) mm, rotated rx -119.62 ry 0 rz 39.38 deg; joints [14.024, -85.39, 129.52, -156.528, 42.165, 133.65, -132.251]
  MoveL 2418 to (82.03, -103.07, 73.83) mm, rotated rx -120.25 ry 0 rz 38.66 deg; joints [14.155, -85.399, 129.586, -156.326, 42.165, 132.891, -131.627]
  MoveL 2419 to (79.28, -104.67, 74.61) mm, rotated rx -120.59 ry 0 rz 37.26 deg; joints [14.258, -85.318, 129.586, -156.207, 42.249, 132.492, -130.243]
  MoveL 2420 to (78.73, -104.93, 74.82) mm, rotated rx -120.59 ry 0 rz 37.26 deg; joints [14.26, -85.27, 129.544, -156.204, 42.25, 132.492, -130.249]
  MoveL 2421 to (77.17, -105.18, 76.07) mm, rotated rx -120.67 ry 0 rz 37.11 deg; joints [14.331, -85.156, 129.544, -156.197, 42.47, 132.448, -130.002]
  MoveL 2422 to (75.93, -104.81, 77.8) mm, rotated rx -121.44 ry 0 rz 36.76 deg; joints [14.56, -84.962, 129.544, -155.945, 42.679, 131.559, -129.692]
  MoveL 2423 to (75.93, -104.84, 77.76) mm, rotated rx -122.01 ry 0 rz 35.98 deg; joints [14.681, -84.973, 129.612, -155.76, 42.679, 130.875, -129.003]
  MoveL 2424 to (72.76, -106.49, 78.55) mm, rotated rx -122.36 ry 0 rz 34.38 deg; joints [14.784, -84.887, 129.612, -155.643, 42.765, 130.47, -127.426]
  MoveL 2425 to (71.88, -107.61, 77.86) mm, rotated rx -121.96 ry 0 rz 32.95 deg; joints [14.69, -85.078, 129.64, -155.643, 42.46, 130.817, -126.125]
  MoveL 2426 to (81.1, -121.85, 88.44) mm, rotated rx -121.96 ry 0 rz 32.95 deg; joints [15.271, -85.671, 129.23, -154.712, 42.46, 129.888, -125.354]
  Set speed (1000.0 mm/s)
  MoveL 2427 to (76.27, -124.33, 89.28) mm, rotated rx -121.88 ry 0 rz 32.18 deg; joints [15.245, -85.425, 129.003, -154.752, 42.46, 130.003, -124.594]
  Set speed (5.0 mm/s)
  MoveL 2428 to (67.23, -109.95, 78.71) mm, rotated rx -121.88 ry 0 rz 32.18 deg; joints [14.667, -84.83, 129.411, -155.679, 42.459, 130.928, -125.368]
  Set speed (16.7 mm/s)
  MoveL 2429 to (66.34, -109.64, 79.86) mm, rotated rx -122.41 ry 0 rz 31.91 deg; joints [14.82, -84.696, 129.411, -155.513, 42.6, 130.331, -125.128]
  MoveL 2430 to (66.4, -109.69, 79.77) mm, rotated rx -122.7 ry 0 rz 30.11 deg; joints [14.922, -84.907, 129.646, -155.356, 42.6, 129.939, -123.384]
  MoveL 2431 to (65.6, -110.87, 78.81) mm, rotated rx -122.26 ry 0 rz 29.53 deg; joints [14.795, -85.021, 129.646, -155.492, 42.478, 130.436, -122.782]
  MoveL 2432 to (65.51, -110.88, 78.88) mm, rotated rx -120.69 ry 0 rz 29.77 deg; joints [14.508, -85.239, 129.646, -155.848, 42.303, 132.183, -122.912]
  MoveL 2433 to (66.11, -110.73, 78.59) mm, rotated rx -120.67 ry 0 rz 29.84 deg; joints [14.493, -85.28, 129.66, -155.848, 42.254, 132.2, -122.998]
  MoveL 2434 to (67.55, -110.49, 77.7) mm, rotated rx -120.26 ry 0 rz 30.45 deg; joints [14.373, -85.379, 129.66, -155.983, 42.148, 132.666, -123.596]
  MoveL 2435 to (76.3, -125.38, 87.78) mm, rotated rx -120.26 ry 0 rz 30.45 deg; joints [14.933, -86.001, 129.267, -155.081, 42.148, 131.755, -122.802]
  Set speed (1000.0 mm/s)
  MoveL 2436 to (81.3, -122.05, 87.96) mm, rotated rx -120.21 ry 0 rz 33.14 deg; joints [14.919, -85.945, 129.212, -155.102, 42.148, 131.825, -125.485]
  Set speed (5.0 mm/s)
  MoveL 2437 to (71.85, -107.58, 77.9) mm, rotated rx -120.21 ry 0 rz 33.14 deg; joints [14.36, -85.322, 129.605, -156.002, 42.148, 132.735, -126.279]
  Set speed (16.7 mm/s)
  MoveL 2438 to (74.32, -106.44, 77.17) mm, rotated rx -119.88 ry 0 rz 34.36 deg; joints [14.262, -85.402, 129.605, -156.115, 42.067, 133.118, -127.474]
  MoveL 2439 to (76.08, -106.16, 75.83) mm, rotated rx -119.88 ry 0 rz 34.36 deg; joints [14.216, -85.556, 129.693, -156.145, 41.978, 133.118, -127.49]
  MoveL 2440 to (76.49, -107.22, 73.91) mm, rotated rx -119.88 ry 0 rz 34.36 deg; joints [14.119, -85.622, 129.694, -156.271, 41.928, 133.187, -127.449]
  MoveL 2441 to (76.36, -107.61, 73.48) mm, rotated rx -119.69 ry 0 rz 34.21 deg; joints [14.061, -85.669, 129.694, -156.336, 41.875, 133.411, -127.297]
  MoveL 2442 to (74.64, -110.62, 70.67) mm, rotated rx -118.61 ry 0 rz 32.99 deg; joints [13.714, -85.928, 129.694, -156.748, 41.604, 134.703, -126.006]
  MoveL 2443 to (74.55, -110.64, 70.76) mm, rotated rx -117.18 ry 0 rz 33.11 deg; joints [13.443, -86.116, 129.694, -157.086, 41.42, 136.31, -126.062]
  MoveL 2444 to (75.37, -110.41, 70.28) mm, rotated rx -116.97 ry 0 rz 33.47 deg; joints [13.377, -86.164, 129.694, -157.164, 41.366, 136.564, -126.406]
  MoveL 2445 to (75.8, -110.29, 70) mm, rotated rx -116.87 ry 0 rz 33.62 deg; joints [13.344, -86.193, 129.694, -157.197, 41.326, 136.678, -126.56]
  MoveL 2446 to (80.22, -109.48, 66.24) mm, rotated rx -115.34 ry 0 rz 35.27 deg; joints [12.854, -86.553, 129.694, -157.762, 40.878, 138.503, -128.187]
  MoveL 2447 to (81.82, -108.86, 65.3) mm, rotated rx -114.8 ry 0 rz 36.17 deg; joints [12.696, -86.638, 129.694, -157.982, 40.813, 139.178, -129.027]
  MoveL 2448 to (82.54, -108.68, 64.7) mm, rotated rx -114.8 ry 0 rz 36.17 deg; joints [12.673, -86.699, 129.724, -157.994, 40.759, 139.178, -129.047]
  MoveL 2449 to (82.97, -108.65, 64.19) mm, rotated rx -114.69 ry 0 rz 36.25 deg; joints [12.626, -86.739, 129.724, -158.04, 40.696, 139.31, -129.145]
  MoveL 2450 to (84.56, -108.68, 62.03) mm, rotated rx -113.77 ry 0 rz 36.79 deg; joints [12.33, -86.932, 129.724, -158.402, 40.459, 140.439, -129.657]
  MoveL 2451 to (85.24, -109.09, 60.34) mm, rotated rx -112.69 ry 0 rz 37.28 deg; joints [12.019, -87.085, 129.724, -158.841, 40.335, 141.797, -130.049]
  MoveL 2452 to (86.29, -108.63, 59.69) mm, rotated rx -112.41 ry 0 rz 37.76 deg; joints [11.93, -87.139, 129.724, -158.954, 40.268, 142.137, -130.514]
  MoveL 2453 to (86.91, -108.41, 59.18) mm, rotated rx -112.41 ry 0 rz 37.76 deg; joints [11.91, -87.191, 129.749, -158.964, 40.217, 142.137, -130.535]
  MoveL 2454 to (87.75, -108.62, 57.54) mm, rotated rx -112.41 ry 0 rz 37.76 deg; joints [11.828, -87.267, 129.749, -159.033, 40.077, 142.167, -130.585]
  MoveL 2455 to (87.87, -108.87, 56.87) mm, rotated rx -112.14 ry 0 rz 37.73 deg; joints [11.737, -87.322, 129.749, -159.148, 40.006, 142.514, -130.556]
  MoveL 2456 to (87.86, -111.36, 51.85) mm, rotated rx -110.24 ry 0 rz 37.14 deg; joints [11.084, -87.691, 129.749, -159.987, 39.517, 144.922, -129.936]
  MoveL 2457 to (87.86, -111.88, 50.72) mm, rotated rx -109.75 ry 0 rz 37 deg; joints [10.922, -87.779, 129.749, -160.197, 39.394, 145.546, -129.799]
  MoveL 2458 to (87.76, -112.25, 50.06) mm, rotated rx -109.75 ry 0 rz 37 deg; joints [10.887, -87.781, 129.742, -160.254, 39.394, 145.586, -129.781]
  MoveL 2459 to (84.83, -117.8, 41.63) mm, rotated rx -106.56 ry 0 rz 35.13 deg; joints [9.765, -88.285, 129.742, -161.809, 38.729, 149.795, -127.821]
  MoveL 2460 to (84.28, -118.46, 40.86) mm, rotated rx -106.56 ry 0 rz 35.13 deg; joints [9.717, -88.251, 129.701, -161.886, 38.729, 149.851, -127.803]
  MoveL 2461 to (83.55, -119.18, 40.28) mm, rotated rx -106.33 ry 0 rz 34.72 deg; joints [9.638, -88.287, 129.701, -161.994, 38.673, 150.152, -127.4]
  MoveL 2462 to (74.71, -125.93, 36.97) mm, rotated rx -105.08 ry 0 rz 30.39 deg; joints [9.191, -88.474, 129.701, -162.617, 38.387, 151.829, -123.079]
  MoveL 2463 to (72.85, -127.36, 35.78) mm, rotated rx -104.54 ry 0 rz 29.31 deg; joints [9.014, -88.565, 129.701, -162.844, 38.213, 152.51, -122.044]
  MoveL 2464 to (72.33, -127.72, 35.56) mm, rotated rx -104.54 ry 0 rz 29.31 deg; joints [8.996, -88.528, 129.663, -162.873, 38.213, 152.531, -122.04]
  MoveL 2465 to (71.7, -128.11, 35.4) mm, rotated rx -104.48 ry 0 rz 29.02 deg; joints [8.974, -88.537, 129.664, -162.904, 38.199, 152.615, -121.752]
  MoveL 2466 to (69.43, -129.62, 34.29) mm, rotated rx -104.01 ry 0 rz 27.81 deg; joints [8.813, -88.616, 129.664, -163.113, 38.044, 153.23, -120.584]
  MoveL 2467 to (70.26, -129.64, 32.62) mm, rotated rx -102.47 ry 0 rz 27.48 deg; joints [8.389, -88.843, 129.664, -163.643, 37.575, 155.115, -120.421]
  MoveL 2468 to (70.31, -129.74, 32.11) mm, rotated rx -102.27 ry 0 rz 27.48 deg; joints [8.318, -88.868, 129.664, -163.747, 37.533, 155.387, -120.426]
  MoveL 2469 to (69.83, -130.42, 30.36) mm, rotated rx -102.27 ry 0 rz 27.48 deg; joints [8.222, -88.859, 129.643, -163.908, 37.533, 155.505, -120.393]
  MoveL 2470 to (67.3, -132.41, 27.29) mm, rotated rx -101.08 ry 0 rz 26.26 deg; joints [7.795, -88.998, 129.643, -164.534, 37.285, 157.133, -119.198]
  MoveL 2471 to (65.83, -133.29, 26.58) mm, rotated rx -101.08 ry 0 rz 26.26 deg; joints [7.744, -88.896, 129.541, -164.62, 37.285, 157.198, -119.189]
  MoveL 2472 to (64.21, -134, 26.97) mm, rotated rx -101.08 ry 0 rz 26.13 deg; joints [7.753, -88.793, 129.453, -164.613, 37.306, 157.198, -119.053]
  MoveL 2473 to (63.32, -134.29, 27.58) mm, rotated rx -101.32 ry 0 rz 25.77 deg; joints [7.836, -88.766, 129.453, -164.49, 37.354, 156.877, -118.688]
  Set speed (1000.0 mm/s)
  MoveL 2474 to (63.32, -134.29, 27.58) mm, rotated rx -101.32 ry 0 rz 25.77 deg; joints [7.836, -88.766, 129.453, -164.49, 37.354, 156.877, -118.688]
  MoveL 2475 to (105.95, -222.6, 47.2) mm, rotated rx -101.32 ry 0 rz 25.77 deg; joints [9.228, -93.555, 128.705, -162.1, 37.354, 154.053, -113.566]
  Call onMillingEarth_Retract
  Call onMillingEarth_Finish

--- program Prog2 ---
